LIN {X 0,Y 482.616,Z 304.958,A -85,B 0,C 180,E1 -7446.836,E2 -7446.836} C_VEL
LIN {X 0,Y 483.015,Z 308.734,A -85,B 0,C 180,E1 -7446.916,E2 -7446.916} C_VEL
LIN {X 0,Y 482.104,Z 314.511,A -85,B 0,C 180,E1 -7446.961,E2 -7446.961} C_VEL
LIN {X 0,Y 476.671,Z 329.767,A -85,B 0,C 180,E1 -7446.925,E2 -7446.925} C_VEL
LIN {X 0,Y 475.779,Z 335.739,A -85,B 0,C 180,E1 -7446.975,E2 -7446.975} C_VEL
LIN {X 0,Y 474.805,Z 416.673,A -85,B 0,C 180,E1 -7448.224,E2 -7448.224} C_VEL
LIN {X 0,Y 474.407,Z 451.66,A -85,B 0,C 180,E1 -7448.789,E2 -7448.789} C_VEL
LIN {X 0,Y 473.978,Z 467.204,A -85,B 0,C 180,E1 -7449.21,E2 -7449.21} C_VEL
LIN {X 0,Y 473.417,Z 481.814,A -85,B 0,C 180,E1 -7449.78,E2 -7449.78} C_VEL
LIN {X 0,Y 472.73,Z 495.057,A -85,B 0,C 180,E1 -7450.457,E2 -7450.457} C_VEL
LIN {X 0,Y 472.006,Z 508.633,A -85,B 0,C 180,E1 -7451.329,E2 -7451.329} C_VEL
LIN {X 0,Y 471.129,Z 521.115,A -85,B 0,C 180,E1 -7452.305,E2 -7452.305} C_VEL
LIN {X 0,Y 470.287,Z 533.744,A -85,B 0,C 180,E1 -7453.504,E2 -7453.504} C_VEL
LIN {X 0,Y 469.473,Z 545.188,A -85,B 0,C 180,E1 -7454.812,E2 -7454.812} C_VEL
LIN {X 0,Y 468.777,Z 554.815,A -85,B 0,C 180,E1 -7456.12,E2 -7456.12} C_VEL
LIN {X 0,Y 468.14,Z 563.629,A -85,B 0,C 180,E1 -7457.535,E2 -7457.535} C_VEL
LIN {X 0,Y 467.659,Z 572.092,A -85,B 0,C 180,E1 -7459.172,E2 -7459.172} C_VEL
LIN {X 0,Y 467.25,Z 579.415,A -85,B 0,C 180,E1 -7460.913,E2 -7460.913} C_VEL
LIN {X 0,Y 466.977,Z 585.225,A -85,B 0,C 180,E1 -7462.65,E2 -7462.65} C_VEL
LIN {X 0,Y 466.904,Z 588.661,A -85,B 0,C 180,E1 -7463.951,E2 -7463.951} C_VEL
LIN {X 0,Y 466.715,Z 592.15,A -85,B 0,C 180,E1 -7465.682,E2 -7465.682} C_VEL
LIN {X 0,Y 466.698,Z 594.456,A -85,B 0,C 180,E1 -7467.41,E2 -7467.41} C_VEL
LIN {X 0,Y 466.617,Z 595.638,A -85,B 0,C 180,E1 -7469.137,E2 -7469.137} C_VEL
LIN {X 0,Y 466.618,Z 595.656,A -85,B 0,C 180,E1 -7470.863,E2 -7470.863} C_VEL
LIN {X 0,Y 466.698,Z 594.543,A -85,B 0,C 180,E1 -7472.589,E2 -7472.589} C_VEL
LIN {X 0,Y 466.714,Z 592.306,A -85,B 0,C 180,E1 -7474.318,E2 -7474.318} C_VEL
LIN {X 0,Y 466.896,Z 588.882,A -85,B 0,C 180,E1 -7476.048,E2 -7476.048} C_VEL
LIN {X 0,Y 467.024,Z 584.198,A -85,B 0,C 180,E1 -7477.783,E2 -7477.783} C_VEL
LIN {X 0,Y 467.297,Z 578.125,A -85,B 0,C 180,E1 -7479.522,E2 -7479.522} C_VEL
LIN {X 0,Y 467.817,Z 570.471,A -85,B 0,C 180,E1 -7481.262,E2 -7481.262} C_VEL
LIN {X 0,Y 468.265,Z 562.094,A -85,B 0,C 180,E1 -7482.827,E2 -7482.827} C_VEL
LIN {X 0,Y 468.995,Z 552.473,A -85,B 0,C 180,E1 -7484.315,E2 -7484.315} C_VEL
LIN {X 0,Y 469.695,Z 542.383,A -85,B 0,C 180,E1 -7485.624,E2 -7485.624} C_VEL
LIN {X 0,Y 470.399,Z 532.32,A -85,B 0,C 180,E1 -7486.732,E2 -7486.732} C_VEL
LIN {X 0,Y 471.236,Z 519.597,A -85,B 0,C 180,E1 -7487.914,E2 -7487.914} C_VEL
LIN {X 0,Y 472.123,Z 506.782,A -85,B 0,C 180,E1 -7488.891,E2 -7488.891} C_VEL
LIN {X 0,Y 472.878,Z 492.726,A -85,B 0,C 180,E1 -7489.762,E2 -7489.762} C_VEL
LIN {X 0,Y 473.588,Z 477.794,A -85,B 0,C 180,E1 -7490.48,E2 -7490.48} C_VEL
LIN {X 0,Y 474.103,Z 462.506,A -85,B 0,C 180,E1 -7491.024,E2 -7491.024} C_VEL
LIN {X 0,Y 474.465,Z 448.708,A -85,B 0,C 180,E1 -7491.358,E2 -7491.358} C_VEL
LIN {X 0,Y 476.043,Z 314.849,A -85,B 0,C 180,E1 -7493.441,E2 -7493.441} C_VEL
LIN {X 0,Y 475.999,Z 305.711,A -85,B 0,C 180,E1 -7493.591,E2 -7493.591} C_VEL
LIN {X 0,Y 472.887,Z 293.254,A -85,B 0,C 180,E1 -7493.96,E2 -7493.96} C_VEL
LIN {X 0,Y 470.172,Z 286.418,A -85,B 0,C 180,E1 -7494.243,E2 -7494.243} C_VEL
LIN {X 0,Y 467.576,Z 274.869,A -85,B 0,C 180,E1 -7496.501,E2 -7496.501} C_VEL
LIN {X 0,Y 467.531,Z 274.875,A -85,B 0,C 180,E1 -7499.739,E2 -7499.739} C_VEL
LIN {X 0,Y 467.547,Z 274.874,A -85,B 0,C 180,E1 -7502.761,E2 -7502.761} C_VEL
LIN {X 0,Y 467.541,Z 274.867,A -85,B 0,C 180,E1 -7505.89,E2 -7505.89} C_VEL
LIN {X 0,Y 467.541,Z 274.873,A -85,B 0,C 180,E1 -7509.148,E2 -7509.148} C_VEL
LIN {X 0,Y 467.556,Z 274.867,A -85,B 0,C 180,E1 -7511.405,E2 -7511.405} C_VEL
LIN {X 0,Y 467.56,Z 274.87,A -85,B 0,C 180,E1 -7515.052,E2 -7515.052} C_VEL
LIN {X 0,Y 467.547,Z 274.863,A -85,B 0,C 180,E1 -7518.727,E2 -7518.727} C_VEL
LIN {X 0,Y 467.531,Z 274.868,A -85,B 0,C 180,E1 -7521.952,E2 -7521.952} C_VEL
LIN {X 0,Y 467.538,Z 274.868,A -85,B 0,C 180,E1 -7525.165,E2 -7525.165} C_VEL
LIN {X 0,Y 467.54,Z 274.871,A -85,B 0,C 180,E1 -7528.257,E2 -7528.257} C_VEL
LIN {X 0,Y 467.522,Z 274.87,A -85,B 0,C 180,E1 -7531.247,E2 -7531.247} C_VEL
LIN {X 0,Y 467.574,Z 274.868,A -85,B 0,C 180,E1 -7534.401,E2 -7534.401} C_VEL
LIN {X 0,Y 467.548,Z 274.866,A -85,B 0,C 180,E1 -7536.994,E2 -7536.994} C_VEL
LIN {X 0,Y 467.586,Z 274.862,A -85,B 0,C 180,E1 -7539.775,E2 -7539.775} C_VEL
LIN {X 0,Y 467.555,Z 274.871,A -85,B 0,C 180,E1 -7542.505,E2 -7542.505} C_VEL
LIN {X 0,Y 467.585,Z 274.858,A -85,B 0,C 180,E1 -7545.196,E2 -7545.196} C_VEL
LIN {X 0,Y 467.655,Z 274.854,A -85,B 0,C 180,E1 -7547.854,E2 -7547.854} C_VEL
LIN {X 0,Y 467.634,Z 274.851,A -85,B 0,C 180,E1 -7551.356,E2 -7551.356} C_VEL
LIN {X 0,Y 467.693,Z 274.852,A -85,B 0,C 180,E1 -7553.962,E2 -7553.962} C_VEL
LIN {X 0,Y 467.846,Z 274.828,A -85,B 0,C 180,E1 -7557.417,E2 -7557.417} C_VEL
LIN {X 0,Y 467.847,Z 274.834,A -85,B 0,C 180,E1 -7560,E2 -7560} C_VEL
LIN {X 0,Y 467.819,Z 274.835,A -85,B 0,C 180,E1 -7562.583,E2 -7562.583} C_VEL
LIN {X 0,Y 467.71,Z 274.847,A -85,B 0,C 180,E1 -7566.038,E2 -7566.038} C_VEL
LIN {X 0,Y 467.662,Z 274.853,A -85,B 0,C 180,E1 -7568.643,E2 -7568.643} C_VEL
LIN {X 0,Y 467.655,Z 274.859,A -85,B 0,C 180,E1 -7572.145,E2 -7572.145} C_VEL
LIN {X 0,Y 467.637,Z 274.855,A -85,B 0,C 180,E1 -7575.695,E2 -7575.695} C_VEL
LIN {X 0,Y 467.62,Z 274.857,A -85,B 0,C 180,E1 -7579.308,E2 -7579.308} C_VEL
LIN {X 0,Y 467.533,Z 274.873,A -85,B 0,C 180,E1 -7582.074,E2 -7582.074} C_VEL
LIN {X 0,Y 467.581,Z 274.849,A -85,B 0,C 180,E1 -7584.888,E2 -7584.888} C_VEL
LIN {X 0,Y 467.578,Z 274.865,A -85,B 0,C 180,E1 -7587.772,E2 -7587.772} C_VEL
LIN {X 0,Y 467.566,Z 274.859,A -85,B 0,C 180,E1 -7591.045,E2 -7591.045} C_VEL
LIN {X 0,Y 467.587,Z 274.864,A -85,B 0,C 180,E1 -7594.242,E2 -7594.242} C_VEL
LIN {X 0,Y 467.546,Z 274.863,A -85,B 0,C 180,E1 -7597.186,E2 -7597.186} C_VEL
LIN {X 0,Y 467.576,Z 274.864,A -85,B 0,C 180,E1 -7600.265,E2 -7600.265} C_VEL
LIN {X 0,Y 467.585,Z 274.862,A -85,B 0,C 180,E1 -7602.567,E2 -7602.567} C_VEL
LIN {X 0,Y 467.564,Z 274.866,A -85,B 0,C 180,E1 -7605.053,E2 -7605.053} C_VEL
LIN {X 0,Y 467.587,Z 274.865,A -85,B 0,C 180,E1 -7607.44,E2 -7607.44} C_VEL
LIN {X 0,Y 467.581,Z 274.864,A -85,B 0,C 180,E1 -7610.855,E2 -7610.855} C_VEL
LIN {X 0,Y 467.561,Z 274.868,A -85,B 0,C 180,E1 -7614.261,E2 -7614.261} C_VEL
LIN {X 0,Y 467.581,Z 274.868,A -85,B 0,C 180,E1 -7617.321,E2 -7617.321} C_VEL
LIN {X 0,Y 467.582,Z 274.98,A -85,B 0,C 180,E1 -7619.153,E2 -7619.153} C_VEL
LIN {X 0,Y 471.016,Z 288.782,A -85,B 0,C 180,E1 -7621.48,E2 -7621.48} C_VEL
LIN {X 0,Y 472.395,Z 295.297,A -85,B 0,C 180,E1 -7622.536,E2 -7622.536} C_VEL
LIN {X 0,Y 471.328,Z 315.414,A -85,B 0,C 180,E1 -7625.446,E2 -7625.446} C_VEL
LIN {X 0,Y 471.122,Z 318.255,A -85,B 0,C 180,E1 -7625.853,E2 -7625.853} C_VEL
LIN {X 0,Y 475.844,Z 343.181,A -85,B 0,C 180,E1 -7626.514,E2 -7626.514} C_VEL
LIN {X 0,Y 474.196,Z 484.206,A -85,B 0,C 180,E1 -7628.709,E2 -7628.709} C_VEL
LIN {X 0,Y 473.7,Z 499.79,A -85,B 0,C 180,E1 -7629.113,E2 -7629.113} C_VEL
LIN {X 0,Y 473.008,Z 515.238,A -85,B 0,C 180,E1 -7629.698,E2 -7629.698} C_VEL
LIN {X 0,Y 472.193,Z 529.814,A -85,B 0,C 180,E1 -7630.435,E2 -7630.435} C_VEL
LIN {X 0,Y 471.378,Z 543.34,A -85,B 0,C 180,E1 -7631.304,E2 -7631.304} C_VEL
LIN {X 0,Y 470.541,Z 555.818,A -85,B 0,C 180,E1 -7632.283,E2 -7632.283} C_VEL
LIN {X 0,Y 469.628,Z 568.514,A -85,B 0,C 180,E1 -7633.481,E2 -7633.481} C_VEL
LIN {X 0,Y 468.867,Z 580.057,A -85,B 0,C 180,E1 -7634.793,E2 -7634.793} C_VEL
LIN {X 0,Y 468.278,Z 589.779,A -85,B 0,C 180,E1 -7636.106,E2 -7636.106} C_VEL
LIN {X 0,Y 467.631,Z 599.448,A -85,B 0,C 180,E1 -7637.655,E2 -7637.655} C_VEL
LIN {X 0,Y 467.34,Z 607.294,A -85,B 0,C 180,E1 -7639.166,E2 -7639.166} C_VEL
LIN {X 0,Y 466.956,Z 614.727,A -85,B 0,C 180,E1 -7640.908,E2 -7640.908} C_VEL
LIN {X 0,Y 466.811,Z 620.631,A -85,B 0,C 180,E1 -7642.648,E2 -7642.648} C_VEL
LIN {X 0,Y 466.705,Z 624.139,A -85,B 0,C 180,E1 -7643.95,E2 -7643.95} C_VEL
LIN {X 0,Y 466.616,Z 627.685,A -85,B 0,C 180,E1 -7645.681,E2 -7645.681} C_VEL
LIN {X 0,Y 466.656,Z 630.021,A -85,B 0,C 180,E1 -7647.411,E2 -7647.411} C_VEL
LIN {X 0,Y 466.617,Z 631.194,A -85,B 0,C 180,E1 -7649.137,E2 -7649.137} C_VEL
LIN {X 0,Y 466.617,Z 631.193,A -85,B 0,C 180,E1 -7650.863,E2 -7650.863} C_VEL
LIN {X 0,Y 466.656,Z 630.016,A -85,B 0,C 180,E1 -7652.59,E2 -7652.59} C_VEL
LIN {X 0,Y 466.616,Z 627.679,A -85,B 0,C 180,E1 -7654.319,E2 -7654.319} C_VEL
LIN {X 0,Y 466.696,Z 624.137,A -85,B 0,C 180,E1 -7656.051,E2 -7656.051} C_VEL
LIN {X 0,Y 466.827,Z 619.299,A -85,B 0,C 180,E1 -7657.788,E2 -7657.788} C_VEL
LIN {X 0,Y 467.001,Z 613.033,A -85,B 0,C 180,E1 -7659.529,E2 -7659.529} C_VEL
LIN {X 0,Y 467.41,Z 605.171,A -85,B 0,C 180,E1 -7661.273,E2 -7661.273} C_VEL
LIN {X 0,Y 467.842,Z 596.762,A -85,B 0,C 180,E1 -7662.81,E2 -7662.81} C_VEL
LIN {X 0,Y 468.466,Z 586.744,A -85,B 0,C 180,E1 -7664.332,E2 -7664.332} C_VEL
LIN {X 0,Y 469.144,Z 576.454,A -85,B 0,C 180,E1 -7665.644,E2 -7665.644} C_VEL
LIN {X 0,Y 470.042,Z 564.048,A -85,B 0,C 180,E1 -7666.968,E2 -7666.968} C_VEL
LIN {X 0,Y 470.895,Z 550.568,A -85,B 0,C 180,E1 -7668.153,E2 -7668.153} C_VEL
LIN {X 0,Y 471.779,Z 536.906,A -85,B 0,C 180,E1 -7669.132,E2 -7669.132} C_VEL
LIN {X 0,Y 472.584,Z 522.762,A -85,B 0,C 180,E1 -7669.945,E2 -7669.945} C_VEL
LIN {X 0,Y 473.305,Z 507.927,A -85,B 0,C 180,E1 -7670.605,E2 -7670.605} C_VEL
LIN {X 0,Y 473.946,Z 492.295,A -85,B 0,C 180,E1 -7671.104,E2 -7671.104} C_VEL
LIN {X 0,Y 474.32,Z 476.367,A -85,B 0,C 180,E1 -7671.428,E2 -7671.428} C_VEL
LIN {X 0,Y 475.826,Z 343.138,A -85,B 0,C 180,E1 -7673.485,E2 -7673.485} C_VEL
LIN {X 0,Y 471.104,Z 318.257,A -85,B 0,C 180,E1 -7674.145,E2 -7674.145} C_VEL
LIN {X 0,Y 472.319,Z 298.282,A -85,B 0,C 180,E1 -7677.022,E2 -7677.022} C_VEL
LIN {X 0,Y 472.405,Z 295.266,A -85,B 0,C 180,E1 -7677.464,E2 -7677.464} C_VEL
LIN {X 0,Y 469.063,Z 280.585,A -85,B 0,C 180,E1 -7679.88,E2 -7679.88} C_VEL
LIN {X 0,Y 467.56,Z 274.867,A -85,B 0,C 180,E1 -7680.878,E2 -7680.878} C_VEL
LIN {X 0,Y 467.588,Z 274.866,A -85,B 0,C 180,E1 -7683.789,E2 -7683.789} C_VEL
LIN {X 0,Y 467.55,Z 274.867,A -85,B 0,C 180,E1 -7687.187,E2 -7687.187} C_VEL
LIN {X 0,Y 467.574,Z 274.863,A -85,B 0,C 180,E1 -7690.266,E2 -7690.266} C_VEL
LIN {X 0,Y 467.551,Z 274.867,A -85,B 0,C 180,E1 -7693.746,E2 -7693.746} C_VEL
LIN {X 0,Y 467.554,Z 274.865,A -85,B 0,C 180,E1 -7696.255,E2 -7696.255} C_VEL
LIN {X 0,Y 467.581,Z 274.865,A -85,B 0,C 180,E1 -7698.724,E2 -7698.724} C_VEL
LIN {X 0,Y 467.565,Z 274.868,A -85,B 0,C 180,E1 -7701.956,E2 -7701.956} C_VEL
LIN {X 0,Y 467.566,Z 274.862,A -85,B 0,C 180,E1 -7705.168,E2 -7705.168} C_VEL
LIN {X 0,Y 467.587,Z 274.865,A -85,B 0,C 180,E1 -7708.26,E2 -7708.26} C_VEL
LIN {X 0,Y 467.559,Z 274.862,A -85,B 0,C 180,E1 -7711.249,E2 -7711.249} C_VEL
LIN {X 0,Y 467.584,Z 274.864,A -85,B 0,C 180,E1 -7714.159,E2 -7714.159} C_VEL
LIN {X 0,Y 467.58,Z 274.858,A -85,B 0,C 180,E1 -7716.996,E2 -7716.996} C_VEL
LIN {X 0,Y 467.626,Z 274.86,A -85,B 0,C 180,E1 -7719.777,E2 -7719.777} C_VEL
LIN {X 0,Y 467.6,Z 274.863,A -85,B 0,C 180,E1 -7722.507,E2 -7722.507} C_VEL
LIN {X 0,Y 467.609,Z 274.856,A -85,B 0,C 180,E1 -7725.197,E2 -7725.197} C_VEL
LIN {X 0,Y 467.662,Z 274.858,A -85,B 0,C 180,E1 -7727.855,E2 -7727.855} C_VEL
LIN {X 0,Y 467.662,Z 274.854,A -85,B 0,C 180,E1 -7731.357,E2 -7731.357} C_VEL
LIN {X 0,Y 467.708,Z 274.851,A -85,B 0,C 180,E1 -7733.962,E2 -7733.962} C_VEL
LIN {X 0,Y 467.818,Z 274.832,A -85,B 0,C 180,E1 -7737.417,E2 -7737.417} C_VEL
LIN {X 0,Y 467.854,Z 274.833,A -85,B 0,C 180,E1 -7740,E2 -7740} C_VEL
LIN {X 0,Y 467.827,Z 274.831,A -85,B 0,C 180,E1 -7742.583,E2 -7742.583} C_VEL
LIN {X 0,Y 467.699,Z 274.849,A -85,B 0,C 180,E1 -7746.038,E2 -7746.038} C_VEL
LIN {X 0,Y 467.64,Z 274.855,A -85,B 0,C 180,E1 -7748.644,E2 -7748.644} C_VEL
LIN {X 0,Y 467.661,Z 274.855,A -85,B 0,C 180,E1 -7752.145,E2 -7752.145} C_VEL
LIN {X 0,Y 467.617,Z 274.862,A -85,B 0,C 180,E1 -7755.696,E2 -7755.696} C_VEL
LIN {X 0,Y 467.577,Z 274.86,A -85,B 0,C 180,E1 -7758.748,E2 -7758.748} C_VEL
LIN {X 0,Y 467.563,Z 274.869,A -85,B 0,C 180,E1 -7761.261,E2 -7761.261} C_VEL
LIN {X 0,Y 467.552,Z 274.869,A -85,B 0,C 180,E1 -7763.945,E2 -7763.945} C_VEL
LIN {X 0,Y 467.529,Z 274.865,A -85,B 0,C 180,E1 -7766.806,E2 -7766.806} C_VEL
LIN {X 0,Y 467.513,Z 274.873,A -85,B 0,C 180,E1 -7769.741,E2 -7769.741} C_VEL
LIN {X 0,Y 467.551,Z 274.866,A -85,B 0,C 180,E1 -7772.761,E2 -7772.761} C_VEL
LIN {X 0,Y 467.541,Z 274.868,A -85,B 0,C 180,E1 -7775.891,E2 -7775.891} C_VEL
LIN {X 0,Y 467.529,Z 274.871,A -85,B 0,C 180,E1 -7779.15,E2 -7779.15} C_VEL
LIN {X 0,Y 467.552,Z 274.87,A -85,B 0,C 180,E1 -7781.406,E2 -7781.406} C_VEL
LIN {X 0,Y 467.532,Z 274.871,A -85,B 0,C 180,E1 -7784.952,E2 -7784.952} C_VEL
LIN {X 0,Y 467.55,Z 274.866,A -85,B 0,C 180,E1 -7788.594,E2 -7788.594} C_VEL
LIN {X 0,Y 467.535,Z 274.868,A -85,B 0,C 180,E1 -7791.952,E2 -7791.952} C_VEL
LIN {X 0,Y 467.543,Z 274.87,A -85,B 0,C 180,E1 -7795.165,E2 -7795.165} C_VEL
LIN {X 0,Y 467.544,Z 274.867,A -85,B 0,C 180,E1 -7798.256,E2 -7798.256} C_VEL
LIN {X 0,Y 467.527,Z 274.876,A -85,B 0,C 180,E1 -7801.247,E2 -7801.247} C_VEL
LIN {X 0,Y 467.57,Z 274.908,A -85,B 0,C 180,E1 -7803.618,E2 -7803.618} C_VEL
LIN {X 0,Y 470.221,Z 286.501,A -85,B 0,C 180,E1 -7805.868,E2 -7805.868} C_VEL
LIN {X 0,Y 473.542,Z 295.441,A -85,B 0,C 180,E1 -7806.204,E2 -7806.204} C_VEL
LIN {X 0,Y 476.129,Z 307.183,A -85,B 0,C 180,E1 -7806.532,E2 -7806.532} C_VEL
LIN {X 0,Y 475.779,Z 335.739,A -85,B 0,C 180,E1 -7806.975,E2 -7806.975} C_VEL
LIN {X 0,Y 475.114,Z 341.592,A -85,B 0,C 180,E1 -7807.034,E2 -7807.034} C_VEL
LIN {X 0,Y 469.576,Z 360.655,A -85,B 0,C 180,E1 -7807.055,E2 -7807.055} C_VEL
LIN {X 0,Y 468.938,Z 366.506,A -85,B 0,C 180,E1 -7807.117,E2 -7807.117} C_VEL
LIN {X 0,Y 467.811,Z 451.948,A -85,B 0,C 180,E1 -7808.475,E2 -7808.475} C_VEL
LIN {X 0,Y 467.371,Z 467.458,A -85,B 0,C 180,E1 -7808.902,E2 -7808.902} C_VEL
LIN {X 0,Y 466.758,Z 482.247,A -85,B 0,C 180,E1 -7809.486,E2 -7809.486} C_VEL
LIN {X 0,Y 465.949,Z 497.227,A -85,B 0,C 180,E1 -7810.276,E2 -7810.276} C_VEL
LIN {X 0,Y 465.169,Z 510.471,A -85,B 0,C 180,E1 -7811.158,E2 -7811.158} C_VEL
LIN {X 0,Y 464.218,Z 523.927,A -85,B 0,C 180,E1 -7812.261,E2 -7812.261} C_VEL
LIN {X 0,Y 463.314,Z 536.125,A -85,B 0,C 180,E1 -7813.475,E2 -7813.475} C_VEL
LIN {X 0,Y 462.476,Z 547.228,A -85,B 0,C 180,E1 -7814.802,E2 -7814.802} C_VEL
LIN {X 0,Y 461.647,Z 558.012,A -85,B 0,C 180,E1 -7816.351,E2 -7816.351} C_VEL
LIN {X 0,Y 461.053,Z 566.951,A -85,B 0,C 180,E1 -7817.901,E2 -7817.901} C_VEL
LIN {X 0,Y 460.499,Z 574.361,A -85,B 0,C 180,E1 -7819.447,E2 -7819.447} C_VEL
LIN {X 0,Y 460.137,Z 581.283,A -85,B 0,C 180,E1 -7821.214,E2 -7821.214} C_VEL
LIN {X 0,Y 459.849,Z 586.724,A -85,B 0,C 180,E1 -7822.977,E2 -7822.977} C_VEL
LIN {X 0,Y 459.701,Z 590.83,A -85,B 0,C 180,E1 -7824.736,E2 -7824.736} C_VEL
LIN {X 0,Y 459.683,Z 593.715,A -85,B 0,C 180,E1 -7826.493,E2 -7826.493} C_VEL
LIN {X 0,Y 459.571,Z 595.456,A -85,B 0,C 180,E1 -7828.247,E2 -7828.247} C_VEL
LIN {X 0,Y 459.528,Z 596.066,A -85,B 0,C 180,E1 -7830,E2 -7830} C_VEL
LIN {X 0,Y 459.572,Z 595.508,A -85,B 0,C 180,E1 -7831.752,E2 -7831.752} C_VEL
LIN {X 0,Y 459.683,Z 593.836,A -85,B 0,C 180,E1 -7833.506,E2 -7833.506} C_VEL
LIN {X 0,Y 459.697,Z 591.017,A -85,B 0,C 180,E1 -7835.263,E2 -7835.263} C_VEL
LIN {X 0,Y 459.844,Z 586.976,A -85,B 0,C 180,E1 -7837.023,E2 -7837.023} C_VEL
LIN {X 0,Y 460.125,Z 581.614,A -85,B 0,C 180,E1 -7838.785,E2 -7838.785} C_VEL
LIN {X 0,Y 460.474,Z 574.782,A -85,B 0,C 180,E1 -7840.553,E2 -7840.553} C_VEL
LIN {X 0,Y 461.015,Z 567.425,A -85,B 0,C 180,E1 -7842.099,E2 -7842.099} C_VEL
LIN {X 0,Y 461.626,Z 558.564,A -85,B 0,C 180,E1 -7843.649,E2 -7843.649} C_VEL
LIN {X 0,Y 462.294,Z 549.524,A -85,B 0,C 180,E1 -7844.977,E2 -7844.977} C_VEL
LIN {X 0,Y 463.106,Z 538.855,A -85,B 0,C 180,E1 -7846.305,E2 -7846.305} C_VEL
LIN {X 0,Y 463.984,Z 527.536,A -85,B 0,C 180,E1 -7847.488,E2 -7847.488} C_VEL
LIN {X 0,Y 464.895,Z 514.473,A -85,B 0,C 180,E1 -7848.624,E2 -7848.624} C_VEL
LIN {X 0,Y 465.793,Z 500.42,A -85,B 0,C 180,E1 -7849.616,E2 -7849.616} C_VEL
LIN {X 0,Y 466.545,Z 487.148,A -85,B 0,C 180,E1 -7850.365,E2 -7850.365} C_VEL
LIN {X 0,Y 467.176,Z 472.197,A -85,B 0,C 180,E1 -7851.02,E2 -7851.02} C_VEL
LIN {X 0,Y 467.672,Z 457.345,A -85,B 0,C 180,E1 -7851.487,E2 -7851.487} C_VEL
LIN {X 0,Y 468.002,Z 442.394,A -85,B 0,C 180,E1 -7851.789,E2 -7851.789} C_VEL
LIN {X 0,Y 469.559,Z 315.136,A -85,B 0,C 180,E1 -7853.783,E2 -7853.783} C_VEL
LIN {X 0,Y 469.469,Z 306.681,A -85,B 0,C 180,E1 -7853.927,E2 -7853.927} C_VEL
LIN {X 0,Y 466.833,Z 296.114,A -85,B 0,C 180,E1 -7854.247,E2 -7854.247} C_VEL
LIN {X 0,Y 463.026,Z 286.71,A -85,B 0,C 180,E1 -7854.64,E2 -7854.64} C_VEL
LIN {X 0,Y 460.504,Z 275.751,A -85,B 0,C 180,E1 -7856.818,E2 -7856.818} C_VEL
LIN {X 0,Y 460.509,Z 275.751,A -85,B 0,C 180,E1 -7859.553,E2 -7859.553} C_VEL
LIN {X 0,Y 460.5,Z 275.75,A -85,B 0,C 180,E1 -7862.924,E2 -7862.924} C_VEL
LIN {X 0,Y 460.484,Z 275.746,A -85,B 0,C 180,E1 -7866.012,E2 -7866.012} C_VEL
LIN {X 0,Y 460.49,Z 275.753,A -85,B 0,C 180,E1 -7868.889,E2 -7868.889} C_VEL
LIN {X 0,Y 460.5,Z 275.745,A -85,B 0,C 180,E1 -7871.598,E2 -7871.598} C_VEL
LIN {X 0,Y 460.508,Z 275.745,A -85,B 0,C 180,E1 -7874.589,E2 -7874.589} C_VEL
LIN {X 0,Y 460.468,Z 275.738,A -85,B 0,C 180,E1 -7877.812,E2 -7877.812} C_VEL
LIN {X 0,Y 460.472,Z 275.749,A -85,B 0,C 180,E1 -7880.131,E2 -7880.131} C_VEL
LIN {X 0,Y 460.452,Z 275.736,A -85,B 0,C 180,E1 -7883.468,E2 -7883.468} C_VEL
LIN {X 0,Y 460.498,Z 275.752,A -85,B 0,C 180,E1 -7886.672,E2 -7886.672} C_VEL
LIN {X 0,Y 460.476,Z 275.746,A -85,B 0,C 180,E1 -7889.757,E2 -7889.757} C_VEL
LIN {X 0,Y 460.485,Z 275.749,A -85,B 0,C 180,E1 -7892.75,E2 -7892.75} C_VEL
LIN {X 0,Y 460.509,Z 275.743,A -85,B 0,C 180,E1 -7895.666,E2 -7895.666} C_VEL
LIN {X 0,Y 460.512,Z 275.75,A -85,B 0,C 180,E1 -7898.581,E2 -7898.581} C_VEL
LIN {X 0,Y 460.533,Z 275.735,A -85,B 0,C 180,E1 -7901.308,E2 -7901.308} C_VEL
LIN {X 0,Y 460.544,Z 275.737,A -85,B 0,C 180,E1 -7904.964,E2 -7904.964} C_VEL
LIN {X 0,Y 460.606,Z 275.736,A -85,B 0,C 180,E1 -7908.559,E2 -7908.559} C_VEL
LIN {X 0,Y 460.621,Z 275.73,A -85,B 0,C 180,E1 -7912.107,E2 -7912.107} C_VEL
LIN {X 0,Y 460.669,Z 275.722,A -85,B 0,C 180,E1 -7914.748,E2 -7914.748} C_VEL
LIN {X 0,Y 460.786,Z 275.707,A -85,B 0,C 180,E1 -7917.377,E2 -7917.377} C_VEL
LIN {X 0,Y 460.817,Z 275.709,A -85,B 0,C 180,E1 -7920,E2 -7920} C_VEL
LIN {X 0,Y 460.763,Z 275.714,A -85,B 0,C 180,E1 -7922.623,E2 -7922.623} C_VEL
LIN {X 0,Y 460.675,Z 275.723,A -85,B 0,C 180,E1 -7926.13,E2 -7926.13} C_VEL
LIN {X 0,Y 460.613,Z 275.731,A -85,B 0,C 180,E1 -7928.776,E2 -7928.776} C_VEL
LIN {X 0,Y 460.612,Z 275.734,A -85,B 0,C 180,E1 -7932.445,E2 -7932.445} C_VEL
LIN {X 0,Y 460.599,Z 275.735,A -85,B 0,C 180,E1 -7935.997,E2 -7935.997} C_VEL
LIN {X 0,Y 460.566,Z 275.737,A -85,B 0,C 180,E1 -7939.616,E2 -7939.616} C_VEL
LIN {X 0,Y 460.509,Z 275.744,A -85,B 0,C 180,E1 -7942.429,E2 -7942.429} C_VEL
LIN {X 0,Y 460.547,Z 275.728,A -85,B 0,C 180,E1 -7945.797,E2 -7945.797} C_VEL
LIN {X 0,Y 460.525,Z 275.745,A -85,B 0,C 180,E1 -7948.235,E2 -7948.235} C_VEL
LIN {X 0,Y 460.519,Z 275.738,A -85,B 0,C 180,E1 -7951.283,E2 -7951.283} C_VEL
LIN {X 0,Y 460.531,Z 275.741,A -85,B 0,C 180,E1 -7954.506,E2 -7954.506} C_VEL
LIN {X 0,Y 460.499,Z 275.74,A -85,B 0,C 180,E1 -7957.623,E2 -7957.623} C_VEL
LIN {X 0,Y 460.54,Z 275.741,A -85,B 0,C 180,E1 -7960.27,E2 -7960.27} C_VEL
LIN {X 0,Y 460.497,Z 275.749,A -85,B 0,C 180,E1 -7963.376,E2 -7963.376} C_VEL
LIN {X 0,Y 460.497,Z 275.744,A -85,B 0,C 180,E1 -7966.625,E2 -7966.625} C_VEL
LIN {X 0,Y 460.54,Z 275.74,A -85,B 0,C 180,E1 -7969.731,E2 -7969.731} C_VEL
LIN {X 0,Y 460.499,Z 275.745,A -85,B 0,C 180,E1 -7972.524,E2 -7972.524} C_VEL
LIN {X 0,Y 460.547,Z 275.743,A -85,B 0,C 180,E1 -7975.624,E2 -7975.624} C_VEL
LIN {X 0,Y 460.55,Z 275.859,A -85,B 0,C 180,E1 -7978.81,E2 -7978.81} C_VEL
LIN {X 0,Y 464.005,Z 289.714,A -85,B 0,C 180,E1 -7981.194,E2 -7981.194} C_VEL
LIN {X 0,Y 465.531,Z 296.646,A -85,B 0,C 180,E1 -7982.341,E2 -7982.341} C_VEL
LIN {X 0,Y 464.653,Z 314.306,A -85,B 0,C 180,E1 -7984.944,E2 -7984.944} C_VEL
LIN {X 0,Y 464.355,Z 317.975,A -85,B 0,C 180,E1 -7985.477,E2 -7985.477} C_VEL
LIN {X 0,Y 469.371,Z 345.068,A -85,B 0,C 180,E1 -7986.206,E2 -7986.206} C_VEL
LIN {X 0,Y 467.544,Z 485.275,A -85,B 0,C 180,E1 -7988.42,E2 -7988.42} C_VEL
LIN {X 0,Y 466.978,Z 501.269,A -85,B 0,C 180,E1 -7988.859,E2 -7988.859} C_VEL
LIN {X 0,Y 466.301,Z 515.516,A -85,B 0,C 180,E1 -7989.418,E2 -7989.418} C_VEL
LIN {X 0,Y 465.468,Z 529.546,A -85,B 0,C 180,E1 -7990.14,E2 -7990.14} C_VEL
LIN {X 0,Y 464.615,Z 543.071,A -85,B 0,C 180,E1 -7991.021,E2 -7991.021} C_VEL
LIN {X 0,Y 463.681,Z 555.546,A -85,B 0,C 180,E1 -7992.012,E2 -7992.012} C_VEL
LIN {X 0,Y 462.854,Z 566.577,A -85,B 0,C 180,E1 -7993.057,E2 -7993.057} C_VEL
LIN {X 0,Y 462.08,Z 577.99,A -85,B 0,C 180,E1 -7994.338,E2 -7994.338} C_VEL
LIN {X 0,Y 461.4,Z 588.008,A -85,B 0,C 180,E1 -7995.67,E2 -7995.67} C_VEL
LIN {X 0,Y 460.795,Z 596.68,A -85,B 0,C 180,E1 -7997.022,E2 -7997.022} C_VEL
LIN {X 0,Y 460.354,Z 604.91,A -85,B 0,C 180,E1 -7998.553,E2 -7998.553} C_VEL
LIN {X 0,Y 460.057,Z 610.943,A -85,B 0,C 180,E1 -7999.882,E2 -7999.882} C_VEL
LIN {X 0,Y 459.783,Z 617.587,A -85,B 0,C 180,E1 -8001.651,E2 -8001.651} C_VEL
LIN {X 0,Y 459.664,Z 621.615,A -85,B 0,C 180,E1 -8002.975,E2 -8002.975} C_VEL
LIN {X 0,Y 459.594,Z 625.798,A -85,B 0,C 180,E1 -8004.736,E2 -8004.736} C_VEL
LIN {X 0,Y 459.568,Z 628.731,A -85,B 0,C 180,E1 -8006.493,E2 -8006.493} C_VEL
LIN {X 0,Y 459.539,Z 630.48,A -85,B 0,C 180,E1 -8008.248,E2 -8008.248} C_VEL
LIN {X 0,Y 459.527,Z 631.079,A -85,B 0,C 180,E1 -8010,E2 -8010} C_VEL
LIN {X 0,Y 459.539,Z 630.477,A -85,B 0,C 180,E1 -8011.753,E2 -8011.753} C_VEL
LIN {X 0,Y 459.568,Z 628.725,A -85,B 0,C 180,E1 -8013.507,E2 -8013.507} C_VEL
LIN {X 0,Y 459.592,Z 625.793,A -85,B 0,C 180,E1 -8015.265,E2 -8015.265} C_VEL
LIN {X 0,Y 459.652,Z 621.615,A -85,B 0,C 180,E1 -8017.026,E2 -8017.026} C_VEL
LIN {X 0,Y 459.836,Z 616.081,A -85,B 0,C 180,E1 -8018.792,E2 -8018.792} C_VEL
LIN {X 0,Y 460.198,Z 609.044,A -85,B 0,C 180,E1 -8020.56,E2 -8020.56} C_VEL
LIN {X 0,Y 460.582,Z 600.285,A -85,B 0,C 180,E1 -8022.335,E2 -8022.335} C_VEL
LIN {X 0,Y 461.191,Z 590.991,A -85,B 0,C 180,E1 -8023.888,E2 -8023.888} C_VEL
LIN {X 0,Y 461.83,Z 581.544,A -85,B 0,C 180,E1 -8025.219,E2 -8025.219} C_VEL
LIN {X 0,Y 462.735,Z 569.304,A -85,B 0,C 180,E1 -8026.659,E2 -8026.659} C_VEL
LIN {X 0,Y 463.629,Z 556.827,A -85,B 0,C 180,E1 -8027.877,E2 -8027.877} C_VEL
LIN {X 0,Y 464.521,Z 544.557,A -85,B 0,C 180,E1 -8028.869,E2 -8028.869} C_VEL
LIN {X 0,Y 465.388,Z 531.312,A -85,B 0,C 180,E1 -8029.749,E2 -8029.749} C_VEL
LIN {X 0,Y 466.212,Z 517.055,A -85,B 0,C 180,E1 -8030.506,E2 -8030.506} C_VEL
LIN {X 0,Y 466.89,Z 502.902,A -85,B 0,C 180,E1 -8031.081,E2 -8031.081} C_VEL
LIN {X 0,Y 467.471,Z 487.442,A -85,B 0,C 180,E1 -8031.527,E2 -8031.527} C_VEL
LIN {X 0,Y 467.826,Z 465.331,A -85,B 0,C 180,E1 -8031.915,E2 -8031.915} C_VEL
LIN {X 0,Y 469.256,Z 343.824,A -85,B 0,C 180,E1 -8033.818,E2 -8033.818} C_VEL
LIN {X 0,Y 464.329,Z 317.858,A -85,B 0,C 180,E1 -8034.539,E2 -8034.539} C_VEL
LIN {X 0,Y 465.558,Z 298.23,A -85,B 0,C 180,E1 -8037.415,E2 -8037.415} C_VEL
LIN {X 0,Y 465.223,Z 294.982,A -85,B 0,C 180,E1 -8037.925,E2 -8037.925} C_VEL
LIN {X 0,Y 461.678,Z 280.296,A -85,B 0,C 180,E1 -8040.409,E2 -8040.409} C_VEL
LIN {X 0,Y 460.527,Z 275.742,A -85,B 0,C 180,E1 -8041.225,E2 -8041.225} C_VEL
LIN {X 0,Y 460.534,Z 275.747,A -85,B 0,C 180,E1 -8044.506,E2 -8044.506} C_VEL
LIN {X 0,Y 460.503,Z 275.745,A -85,B 0,C 180,E1 -8047.624,E2 -8047.624} C_VEL
LIN {X 0,Y 460.539,Z 275.739,A -85,B 0,C 180,E1 -8050.269,E2 -8050.269} C_VEL
LIN {X 0,Y 460.511,Z 275.743,A -85,B 0,C 180,E1 -8053.375,E2 -8053.375} C_VEL
LIN {X 0,Y 460.499,Z 275.743,A -85,B 0,C 180,E1 -8056.625,E2 -8056.625} C_VEL
LIN {X 0,Y 460.542,Z 275.74,A -85,B 0,C 180,E1 -8059.732,E2 -8059.732} C_VEL
LIN {X 0,Y 460.5,Z 275.749,A -85,B 0,C 180,E1 -8062.525,E2 -8062.525} C_VEL
LIN {X 0,Y 460.549,Z 275.737,A -85,B 0,C 180,E1 -8065.624,E2 -8065.624} C_VEL
LIN {X 0,Y 460.541,Z 275.74,A -85,B 0,C 180,E1 -8068.745,E2 -8068.745} C_VEL
LIN {X 0,Y 460.555,Z 275.742,A -85,B 0,C 180,E1 -8072.262,E2 -8072.262} C_VEL
LIN {X 0,Y 460.538,Z 275.74,A -85,B 0,C 180,E1 -8074.704,E2 -8074.704} C_VEL
LIN {X 0,Y 460.515,Z 275.74,A -85,B 0,C 180,E1 -8077.572,E2 -8077.572} C_VEL
LIN {X 0,Y 460.572,Z 275.735,A -85,B 0,C 180,E1 -8080.385,E2 -8080.385} C_VEL
LIN {X 0,Y 460.609,Z 275.734,A -85,B 0,C 180,E1 -8084.059,E2 -8084.059} C_VEL
LIN {X 0,Y 460.615,Z 275.734,A -85,B 0,C 180,E1 -8087.666,E2 -8087.666} C_VEL
LIN {X 0,Y 460.614,Z 275.731,A -85,B 0,C 180,E1 -8091.224,E2 -8091.224} C_VEL
LIN {X 0,Y 460.674,Z 275.725,A -85,B 0,C 180,E1 -8093.87,E2 -8093.87} C_VEL
LIN {X 0,Y 460.762,Z 275.711,A -85,B 0,C 180,E1 -8097.377,E2 -8097.377} C_VEL
LIN {X 0,Y 460.823,Z 275.708,A -85,B 0,C 180,E1 -8100,E2 -8100} C_VEL
LIN {X 0,Y 460.772,Z 275.71,A -85,B 0,C 180,E1 -8102.623,E2 -8102.623} C_VEL
LIN {X 0,Y 460.665,Z 275.724,A -85,B 0,C 180,E1 -8106.131,E2 -8106.131} C_VEL
LIN {X 0,Y 460.595,Z 275.733,A -85,B 0,C 180,E1 -8108.777,E2 -8108.777} C_VEL
LIN {X 0,Y 460.614,Z 275.731,A -85,B 0,C 180,E1 -8112.334,E2 -8112.334} C_VEL
LIN {X 0,Y 460.562,Z 275.741,A -85,B 0,C 180,E1 -8115.978,E2 -8115.978} C_VEL
LIN {X 0,Y 460.535,Z 275.737,A -85,B 0,C 180,E1 -8118.886,E2 -8118.886} C_VEL
LIN {X 0,Y 460.513,Z 275.749,A -85,B 0,C 180,E1 -8121.486,E2 -8121.486} C_VEL
LIN {X 0,Y 460.514,Z 275.743,A -85,B 0,C 180,E1 -8124.334,E2 -8124.334} C_VEL
LIN {X 0,Y 460.488,Z 275.741,A -85,B 0,C 180,E1 -8127.249,E2 -8127.249} C_VEL
LIN {X 0,Y 460.482,Z 275.746,A -85,B 0,C 180,E1 -8130.242,E2 -8130.242} C_VEL
LIN {X 0,Y 460.503,Z 275.747,A -85,B 0,C 180,E1 -8133.327,E2 -8133.327} C_VEL
LIN {X 0,Y 460.458,Z 275.748,A -85,B 0,C 180,E1 -8136.531,E2 -8136.531} C_VEL
LIN {X 0,Y 460.477,Z 275.749,A -85,B 0,C 180,E1 -8139.868,E2 -8139.868} C_VEL
LIN {X 0,Y 460.458,Z 275.752,A -85,B 0,C 180,E1 -8142.892,E2 -8142.892} C_VEL
LIN {X 0,Y 460.481,Z 275.747,A -85,B 0,C 180,E1 -8145.834,E2 -8145.834} C_VEL
LIN {X 0,Y 460.501,Z 275.748,A -85,B 0,C 180,E1 -8148.985,E2 -8148.985} C_VEL
LIN {X 0,Y 460.48,Z 275.746,A -85,B 0,C 180,E1 -8152.374,E2 -8152.374} C_VEL
LIN {X 0,Y 460.524,Z 275.74,A -85,B 0,C 180,E1 -8155.621,E2 -8155.621} C_VEL
LIN {X 0,Y 460.506,Z 275.745,A -85,B 0,C 180,E1 -8158.742,E2 -8158.742} C_VEL
LIN {X 0,Y 460.497,Z 275.749,A -85,B 0,C 180,E1 -8161.763,E2 -8161.763} C_VEL
LIN {X 0,Y 460.509,Z 275.832,A -85,B 0,C 180,E1 -8163.303,E2 -8163.303} C_VEL
LIN {X 0,Y 463.1,Z 286.999,A -85,B 0,C 180,E1 -8165.483,E2 -8165.483} C_VEL
LIN {X 0,Y 467.347,Z 297.823,A -85,B 0,C 180,E1 -8165.903,E2 -8165.903} C_VEL
LIN {X 0,Y 469.638,Z 307.787,A -85,B 0,C 180,E1 -8166.193,E2 -8166.193} C_VEL
LIN {X 0,Y 468.938,Z 366.506,A -85,B 0,C 180,E1 -8167.117,E2 -8167.117} C_VEL
LIN {X 0,Y 468.312,Z 372.352,A -85,B 0,C 180,E1 -8167.179,E2 -8167.179} C_VEL
LIN {X 0,Y 462.791,Z 391.409,A -85,B 0,C 180,E1 -8167.203,E2 -8167.203} C_VEL
LIN {X 0,Y 462.062,Z 397.262,A -85,B 0,C 180,E1 -8167.261,E2 -8167.261} C_VEL
LIN {X 0,Y 461.213,Z 452.539,A -85,B 0,C 180,E1 -8168.159,E2 -8168.159} C_VEL
LIN {X 0,Y 460.77,Z 467.466,A -85,B 0,C 180,E1 -8168.574,E2 -8168.574} C_VEL
LIN {X 0,Y 460.154,Z 481.74,A -85,B 0,C 180,E1 -8169.141,E2 -8169.141} C_VEL
LIN {X 0,Y 459.384,Z 495.613,A -85,B 0,C 180,E1 -8169.865,E2 -8169.865} C_VEL
LIN {X 0,Y 458.56,Z 509.187,A -85,B 0,C 180,E1 -8170.76,E2 -8170.76} C_VEL
LIN {X 0,Y 457.604,Z 521.667,A -85,B 0,C 180,E1 -8171.764,E2 -8171.764} C_VEL
LIN {X 0,Y 456.651,Z 534.295,A -85,B 0,C 180,E1 -8172.997,E2 -8172.997} C_VEL
LIN {X 0,Y 455.754,Z 545.738,A -85,B 0,C 180,E1 -8174.344,E2 -8174.344} C_VEL
LIN {X 0,Y 454.964,Z 555.364,A -85,B 0,C 180,E1 -8175.69,E2 -8175.69} C_VEL
LIN {X 0,Y 454.164,Z 564.998,A -85,B 0,C 180,E1 -8177.298,E2 -8177.298} C_VEL
LIN {X 0,Y 453.658,Z 572.64,A -85,B 0,C 180,E1 -8178.834,E2 -8178.834} C_VEL
LIN {X 0,Y 453.17,Z 579.962,A -85,B 0,C 180,E1 -8180.628,E2 -8180.628} C_VEL
LIN {X 0,Y 452.859,Z 585.77,A -85,B 0,C 180,E1 -8182.419,E2 -8182.419} C_VEL
LIN {X 0,Y 452.763,Z 589.205,A -85,B 0,C 180,E1 -8183.762,E2 -8183.762} C_VEL
LIN {X 0,Y 452.542,Z 592.693,A -85,B 0,C 180,E1 -8185.546,E2 -8185.546} C_VEL
LIN {X 0,Y 452.544,Z 594.996,A -85,B 0,C 180,E1 -8187.329,E2 -8187.329} C_VEL
LIN {X 0,Y 452.456,Z 596.178,A -85,B 0,C 180,E1 -8189.11,E2 -8189.11} C_VEL
LIN {X 0,Y 452.457,Z 596.195,A -85,B 0,C 180,E1 -8190.89,E2 -8190.89} C_VEL
LIN {X 0,Y 452.545,Z 595.082,A -85,B 0,C 180,E1 -8192.67,E2 -8192.67} C_VEL
LIN {X 0,Y 452.54,Z 592.846,A -85,B 0,C 180,E1 -8194.453,E2 -8194.453} C_VEL
LIN {X 0,Y 452.752,Z 589.421,A -85,B 0,C 180,E1 -8196.238,E2 -8196.238} C_VEL
LIN {X 0,Y 452.93,Z 584.737,A -85,B 0,C 180,E1 -8198.027,E2 -8198.027} C_VEL
LIN {X 0,Y 453.262,Z 578.664,A -85,B 0,C 180,E1 -8199.82,E2 -8199.82} C_VEL
LIN {X 0,Y 453.864,Z 571.008,A -85,B 0,C 180,E1 -8201.613,E2 -8201.613} C_VEL
LIN {X 0,Y 454.321,Z 563.113,A -85,B 0,C 180,E1 -8203.141,E2 -8203.141} C_VEL
LIN {X 0,Y 455.189,Z 553.01,A -85,B 0,C 180,E1 -8204.759,E2 -8204.759} C_VEL
LIN {X 0,Y 455.981,Z 542.919,A -85,B 0,C 180,E1 -8206.107,E2 -8206.107} C_VEL
LIN {X 0,Y 456.877,Z 531.985,A -85,B 0,C 180,E1 -8207.337,E2 -8207.337} C_VEL
LIN {X 0,Y 457.721,Z 520.128,A -85,B 0,C 180,E1 -8208.462,E2 -8208.462} C_VEL
LIN {X 0,Y 458.726,Z 507.31,A -85,B 0,C 180,E1 -8209.464,E2 -8209.464} C_VEL
LIN {X 0,Y 459.442,Z 495.231,A -85,B 0,C 180,E1 -8210.248,E2 -8210.248} C_VEL
LIN {X 0,Y 460.219,Z 481.066,A -85,B 0,C 180,E1 -8210.979,E2 -8210.979} C_VEL
LIN {X 0,Y 460.808,Z 466.473,A -85,B 0,C 180,E1 -8211.55,E2 -8211.55} C_VEL
LIN {X 0,Y 461.2,Z 451.879,A -85,B 0,C 180,E1 -8211.951,E2 -8211.951} C_VEL
LIN {X 0,Y 462.762,Z 340.849,A -85,B 0,C 180,E1 -8213.731,E2 -8213.731} C_VEL
LIN {X 0,Y 462.99,Z 307.826,A -85,B 0,C 180,E1 -8214.268,E2 -8214.268} C_VEL
LIN {X 0,Y 460.572,Z 298.429,A -85,B 0,C 180,E1 -8214.564,E2 -8214.564} C_VEL
LIN {X 0,Y 455.866,Z 287.079,A -85,B 0,C 180,E1 -8215.038,E2 -8215.038} C_VEL
LIN {X 0,Y 453.469,Z 276.627,A -85,B 0,C 180,E1 -8217.144,E2 -8217.144} C_VEL
LIN {X 0,Y 453.468,Z 276.627,A -85,B 0,C 180,E1 -8219.783,E2 -8219.783} C_VEL
LIN {X 0,Y 453.463,Z 276.626,A -85,B 0,C 180,E1 -8223.184,E2 -8223.184} C_VEL
LIN {X 0,Y 453.439,Z 276.624,A -85,B 0,C 180,E1 -8226.296,E2 -8226.296} C_VEL
LIN {X 0,Y 453.44,Z 276.627,A -85,B 0,C 180,E1 -8229.455,E2 -8229.455} C_VEL
LIN {X 0,Y 453.433,Z 276.625,A -85,B 0,C 180,E1 -8231.929,E2 -8231.929} C_VEL
LIN {X 0,Y 453.473,Z 276.621,A -85,B 0,C 180,E1 -8235.472,E2 -8235.472} C_VEL
LIN {X 0,Y 453.461,Z 276.621,A -85,B 0,C 180,E1 -8239.387,E2 -8239.387} C_VEL
LIN {X 0,Y 453.429,Z 276.616,A -85,B 0,C 180,E1 -8242.808,E2 -8242.808} C_VEL
LIN {X 0,Y 453.451,Z 276.622,A -85,B 0,C 180,E1 -8246.085,E2 -8246.085} C_VEL
LIN {X 0,Y 453.444,Z 276.623,A -85,B 0,C 180,E1 -8249.238,E2 -8249.238} C_VEL
LIN {X 0,Y 453.468,Z 276.623,A -85,B 0,C 180,E1 -8252.293,E2 -8252.293} C_VEL
LIN {X 0,Y 453.463,Z 276.621,A -85,B 0,C 180,E1 -8255.263,E2 -8255.263} C_VEL
LIN {X 0,Y 453.474,Z 276.625,A -85,B 0,C 180,E1 -8258.417,E2 -8258.417} C_VEL
LIN {X 0,Y 453.483,Z 276.615,A -85,B 0,C 180,E1 -8261.007,E2 -8261.007} C_VEL
LIN {X 0,Y 453.515,Z 276.614,A -85,B 0,C 180,E1 -8264.725,E2 -8264.725} C_VEL
LIN {X 0,Y 453.555,Z 276.617,A -85,B 0,C 180,E1 -8268.379,E2 -8268.379} C_VEL
LIN {X 0,Y 453.559,Z 276.604,A -85,B 0,C 180,E1 -8271.086,E2 -8271.086} C_VEL
LIN {X 0,Y 453.627,Z 276.603,A -85,B 0,C 180,E1 -8273.774,E2 -8273.774} C_VEL
LIN {X 0,Y 453.73,Z 276.586,A -85,B 0,C 180,E1 -8277.337,E2 -8277.337} C_VEL
LIN {X 0,Y 453.766,Z 276.587,A -85,B 0,C 180,E1 -8280,E2 -8280} C_VEL
LIN {X 0,Y 453.71,Z 276.592,A -85,B 0,C 180,E1 -8282.663,E2 -8282.663} C_VEL
LIN {X 0,Y 453.641,Z 276.599,A -85,B 0,C 180,E1 -8286.226,E2 -8286.226} C_VEL
LIN {X 0,Y 453.58,Z 276.606,A -85,B 0,C 180,E1 -8288.914,E2 -8288.914} C_VEL
LIN {X 0,Y 453.562,Z 276.611,A -85,B 0,C 180,E1 -8292.529,E2 -8292.529} C_VEL
LIN {X 0,Y 453.543,Z 276.616,A -85,B 0,C 180,E1 -8296.196,E2 -8296.196} C_VEL
LIN {X 0,Y 453.515,Z 276.612,A -85,B 0,C 180,E1 -8299.039,E2 -8299.039} C_VEL
LIN {X 0,Y 453.475,Z 276.627,A -85,B 0,C 180,E1 -8301.836,E2 -8301.836} C_VEL
LIN {X 0,Y 453.498,Z 276.602,A -85,B 0,C 180,E1 -8304.735,E2 -8304.735} C_VEL
LIN {X 0,Y 453.504,Z 276.621,A -85,B 0,C 180,E1 -8307.953,E2 -8307.953} C_VEL
LIN {X 0,Y 453.473,Z 276.614,A -85,B 0,C 180,E1 -8310.76,E2 -8310.76} C_VEL
LIN {X 0,Y 453.476,Z 276.623,A -85,B 0,C 180,E1 -8313.913,E2 -8313.913} C_VEL
LIN {X 0,Y 453.451,Z 276.618,A -85,B 0,C 180,E1 -8317.19,E2 -8317.19} C_VEL
LIN {X 0,Y 453.515,Z 276.617,A -85,B 0,C 180,E1 -8319.447,E2 -8319.447} C_VEL
LIN {X 0,Y 453.461,Z 276.623,A -85,B 0,C 180,E1 -8322.995,E2 -8322.995} C_VEL
LIN {X 0,Y 453.462,Z 276.626,A -85,B 0,C 180,E1 -8325.779,E2 -8325.779} C_VEL
LIN {X 0,Y 453.477,Z 276.618,A -85,B 0,C 180,E1 -8328.209,E2 -8328.209} C_VEL
LIN {X 0,Y 453.493,Z 276.619,A -85,B 0,C 180,E1 -8330.794,E2 -8330.794} C_VEL
LIN {X 0,Y 453.455,Z 276.628,A -85,B 0,C 180,E1 -8333.918,E2 -8333.918} C_VEL
LIN {X 0,Y 453.482,Z 276.625,A -85,B 0,C 180,E1 -8337.152,E2 -8337.152} C_VEL
LIN {X 0,Y 453.497,Z 276.83,A -85,B 0,C 180,E1 -8338.468,E2 -8338.468} C_VEL
LIN {X 0,Y 457.031,Z 290.794,A -85,B 0,C 180,E1 -8340.922,E2 -8340.922} C_VEL
LIN {X 0,Y 458.67,Z 297.99,A -85,B 0,C 180,E1 -8342.139,E2 -8342.139} C_VEL
LIN {X 0,Y 458.311,Z 306.172,A -85,B 0,C 180,E1 -8343.373,E2 -8343.373} C_VEL
LIN {X 0,Y 457.62,Z 317.737,A -85,B 0,C 180,E1 -8345.097,E2 -8345.097} C_VEL
LIN {X 0,Y 462.857,Z 345.858,A -85,B 0,C 180,E1 -8345.867,E2 -8345.867} C_VEL
LIN {X 0,Y 460.98,Z 483.693,A -85,B 0,C 180,E1 -8348.067,E2 -8348.067} C_VEL
LIN {X 0,Y 460.42,Z 499.265,A -85,B 0,C 180,E1 -8348.481,E2 -8348.481} C_VEL
LIN {X 0,Y 459.687,Z 514.86,A -85,B 0,C 180,E1 -8349.089,E2 -8349.089} C_VEL
LIN {X 0,Y 458.779,Z 529.279,A -85,B 0,C 180,E1 -8349.838,E2 -8349.838} C_VEL
LIN {X 0,Y 457.85,Z 542.802,A -85,B 0,C 180,E1 -8350.73,E2 -8350.73} C_VEL
LIN {X 0,Y 456.797,Z 556.575,A -85,B 0,C 180,E1 -8351.847,E2 -8351.847} C_VEL
LIN {X 0,Y 455.752,Z 569.072,A -85,B 0,C 180,E1 -8353.081,E2 -8353.081} C_VEL
LIN {X 0,Y 455.014,Z 579.513,A -85,B 0,C 180,E1 -8354.318,E2 -8354.318} C_VEL
LIN {X 0,Y 454.333,Z 589.234,A -85,B 0,C 180,E1 -8355.671,E2 -8355.671} C_VEL
LIN {X 0,Y 453.627,Z 598.783,A -85,B 0,C 180,E1 -8357.246,E2 -8357.246} C_VEL
LIN {X 0,Y 453.281,Z 606.75,A -85,B 0,C 180,E1 -8358.825,E2 -8358.825} C_VEL
LIN {X 0,Y 452.814,Z 614.183,A -85,B 0,C 180,E1 -8360.621,E2 -8360.621} C_VEL
LIN {X 0,Y 452.646,Z 620.088,A -85,B 0,C 180,E1 -8362.417,E2 -8362.417} C_VEL
LIN {X 0,Y 452.542,Z 623.597,A -85,B 0,C 180,E1 -8363.759,E2 -8363.759} C_VEL
LIN {X 0,Y 452.45,Z 627.144,A -85,B 0,C 180,E1 -8365.546,E2 -8365.546} C_VEL
LIN {X 0,Y 452.501,Z 629.482,A -85,B 0,C 180,E1 -8367.33,E2 -8367.33} C_VEL
LIN {X 0,Y 452.454,Z 630.655,A -85,B 0,C 180,E1 -8369.11,E2 -8369.11} C_VEL
LIN {X 0,Y 452.454,Z 630.654,A -85,B 0,C 180,E1 -8370.89,E2 -8370.89} C_VEL
LIN {X 0,Y 452.501,Z 629.476,A -85,B 0,C 180,E1 -8372.671,E2 -8372.671} C_VEL
LIN {X 0,Y 452.45,Z 627.137,A -85,B 0,C 180,E1 -8374.455,E2 -8374.455} C_VEL
LIN {X 0,Y 452.513,Z 623.484,A -85,B 0,C 180,E1 -8376.287,E2 -8376.287} C_VEL
LIN {X 0,Y 452.671,Z 618.753,A -85,B 0,C 180,E1 -8378.033,E2 -8378.033} C_VEL
LIN {X 0,Y 452.87,Z 612.485,A -85,B 0,C 180,E1 -8379.829,E2 -8379.829} C_VEL
LIN {X 0,Y 453.291,Z 605.714,A -85,B 0,C 180,E1 -8381.402,E2 -8381.402} C_VEL
LIN {X 0,Y 453.761,Z 597.527,A -85,B 0,C 180,E1 -8382.979,E2 -8382.979} C_VEL
LIN {X 0,Y 454.437,Z 587.72,A -85,B 0,C 180,E1 -8384.556,E2 -8384.556} C_VEL
LIN {X 0,Y 455.184,Z 577.698,A -85,B 0,C 180,E1 -8385.906,E2 -8385.906} C_VEL
LIN {X 0,Y 456.022,Z 566.767,A -85,B 0,C 180,E1 -8387.155,E2 -8387.155} C_VEL
LIN {X 0,Y 456.987,Z 553.953,A -85,B 0,C 180,E1 -8388.378,E2 -8388.378} C_VEL
LIN {X 0,Y 457.967,Z 541.165,A -85,B 0,C 180,E1 -8389.382,E2 -8389.382} C_VEL
LIN {X 0,Y 458.917,Z 527.221,A -85,B 0,C 180,E1 -8390.273,E2 -8390.273} C_VEL
LIN {X 0,Y 459.734,Z 513.621,A -85,B 0,C 180,E1 -8390.963,E2 -8390.963} C_VEL
LIN {X 0,Y 460.389,Z 499.168,A -85,B 0,C 180,E1 -8391.522,E2 -8391.522} C_VEL
LIN {X 0,Y 460.99,Z 483.506,A -85,B 0,C 180,E1 -8391.933,E2 -8391.933} C_VEL
LIN {X 0,Y 462.809,Z 346.577,A -85,B 0,C 180,E1 -8394.12,E2 -8394.12} C_VEL
LIN {X 0,Y 462.223,Z 342.081,A -85,B 0,C 180,E1 -8394.227,E2 -8394.227} C_VEL
LIN {X 0,Y 457.6,Z 317.666,A -85,B 0,C 180,E1 -8394.911,E2 -8394.911} C_VEL
LIN {X 0,Y 458.761,Z 299.565,A -85,B 0,C 180,E1 -8397.608,E2 -8397.608} C_VEL
LIN {X 0,Y 457.62,Z 293.362,A -85,B 0,C 180,E1 -8398.635,E2 -8398.635} C_VEL
LIN {X 0,Y 454.749,Z 281.641,A -85,B 0,C 180,E1 -8400.665,E2 -8400.665} C_VEL
LIN {X 0,Y 453.479,Z 276.621,A -85,B 0,C 180,E1 -8401.578,E2 -8401.578} C_VEL
LIN {X 0,Y 453.49,Z 276.623,A -85,B 0,C 180,E1 -8404.778,E2 -8404.778} C_VEL
LIN {X 0,Y 453.462,Z 276.627,A -85,B 0,C 180,E1 -8408.313,E2 -8408.313} C_VEL
LIN {X 0,Y 453.496,Z 276.621,A -85,B 0,C 180,E1 -8410.609,E2 -8410.609} C_VEL
LIN {X 0,Y 453.463,Z 276.626,A -85,B 0,C 180,E1 -8414.222,E2 -8414.222} C_VEL
LIN {X 0,Y 453.465,Z 276.62,A -85,B 0,C 180,E1 -8417.005,E2 -8417.005} C_VEL
LIN {X 0,Y 453.497,Z 276.617,A -85,B 0,C 180,E1 -8419.409,E2 -8419.409} C_VEL
LIN {X 0,Y 453.449,Z 276.626,A -85,B 0,C 180,E1 -8422.228,E2 -8422.228} C_VEL
LIN {X 0,Y 453.49,Z 276.615,A -85,B 0,C 180,E1 -8425.223,E2 -8425.223} C_VEL
LIN {X 0,Y 453.47,Z 276.623,A -85,B 0,C 180,E1 -8428.475,E2 -8428.475} C_VEL
LIN {X 0,Y 453.496,Z 276.614,A -85,B 0,C 180,E1 -8431.287,E2 -8431.287} C_VEL
LIN {X 0,Y 453.508,Z 276.618,A -85,B 0,C 180,E1 -8434.284,E2 -8434.284} C_VEL
LIN {X 0,Y 453.483,Z 276.614,A -85,B 0,C 180,E1 -8437.204,E2 -8437.204} C_VEL
LIN {X 0,Y 453.508,Z 276.619,A -85,B 0,C 180,E1 -8440.066,E2 -8440.066} C_VEL
LIN {X 0,Y 453.502,Z 276.617,A -85,B 0,C 180,E1 -8442.876,E2 -8442.876} C_VEL
LIN {X 0,Y 453.516,Z 276.614,A -85,B 0,C 180,E1 -8445.644,E2 -8445.644} C_VEL
LIN {X 0,Y 453.563,Z 276.607,A -85,B 0,C 180,E1 -8448.379,E2 -8448.379} C_VEL
LIN {X 0,Y 453.582,Z 276.607,A -85,B 0,C 180,E1 -8451.087,E2 -8451.087} C_VEL
LIN {X 0,Y 453.642,Z 276.6,A -85,B 0,C 180,E1 -8453.774,E2 -8453.774} C_VEL
LIN {X 0,Y 453.709,Z 276.589,A -85,B 0,C 180,E1 -8457.337,E2 -8457.337} C_VEL
LIN {X 0,Y 453.772,Z 276.587,A -85,B 0,C 180,E1 -8460,E2 -8460} C_VEL
LIN {X 0,Y 453.719,Z 276.588,A -85,B 0,C 180,E1 -8462.664,E2 -8462.664} C_VEL
LIN {X 0,Y 453.634,Z 276.599,A -85,B 0,C 180,E1 -8466.226,E2 -8466.226} C_VEL
LIN {X 0,Y 453.565,Z 276.609,A -85,B 0,C 180,E1 -8468.914,E2 -8468.914} C_VEL
LIN {X 0,Y 453.569,Z 276.608,A -85,B 0,C 180,E1 -8472.529,E2 -8472.529} C_VEL
LIN {X 0,Y 453.501,Z 276.618,A -85,B 0,C 180,E1 -8476.198,E2 -8476.198} C_VEL
LIN {X 0,Y 453.49,Z 276.616,A -85,B 0,C 180,E1 -8479.027,E2 -8479.027} C_VEL
LIN {X 0,Y 453.473,Z 276.621,A -85,B 0,C 180,E1 -8481.836,E2 -8481.836} C_VEL
LIN {X 0,Y 453.465,Z 276.621,A -85,B 0,C 180,E1 -8484.737,E2 -8484.737} C_VEL
LIN {X 0,Y 453.459,Z 276.61,A -85,B 0,C 180,E1 -8487.941,E2 -8487.941} C_VEL
LIN {X 0,Y 453.45,Z 276.623,A -85,B 0,C 180,E1 -8490.762,E2 -8490.762} C_VEL
LIN {X 0,Y 453.456,Z 276.624,A -85,B 0,C 180,E1 -8493.915,E2 -8493.915} C_VEL
LIN {X 0,Y 453.434,Z 276.628,A -85,B 0,C 180,E1 -8497.192,E2 -8497.192} C_VEL
LIN {X 0,Y 453.467,Z 276.621,A -85,B 0,C 180,E1 -8500.612,E2 -8500.612} C_VEL
LIN {X 0,Y 453.436,Z 276.623,A -85,B 0,C 180,E1 -8504.225,E2 -8504.225} C_VEL
LIN {X 0,Y 453.398,Z 276.632,A -85,B 0,C 180,E1 -8506.997,E2 -8506.997} C_VEL
LIN {X 0,Y 453.466,Z 276.626,A -85,B 0,C 180,E1 -8509.413,E2 -8509.413} C_VEL
LIN {X 0,Y 453.433,Z 276.624,A -85,B 0,C 180,E1 -8512.808,E2 -8512.808} C_VEL
LIN {X 0,Y 453.455,Z 276.621,A -85,B 0,C 180,E1 -8516.085,E2 -8516.085} C_VEL
LIN {X 0,Y 453.448,Z 276.629,A -85,B 0,C 180,E1 -8519.238,E2 -8519.238} C_VEL
LIN {X 0,Y 453.47,Z 276.622,A -85,B 0,C 180,E1 -8522.293,E2 -8522.293} C_VEL
LIN {X 0,Y 453.482,Z 276.749,A -85,B 0,C 180,E1 -8522.981,E2 -8522.981} C_VEL
LIN {X 0,Y 455.938,Z 287.319,A -85,B 0,C 180,E1 -8525.072,E2 -8525.072} C_VEL
LIN {X 0,Y 461.139,Z 300.144,A -85,B 0,C 180,E1 -8525.592,E2 -8525.592} C_VEL
LIN {X 0,Y 463.12,Z 309.434,A -85,B 0,C 180,E1 -8525.859,E2 -8525.859} C_VEL
LIN {X 0,Y 462.062,Z 397.262,A -85,B 0,C 180,E1 -8527.261,E2 -8527.261} C_VEL
LIN {X 0,Y 461.322,Z 403.108,A -85,B 0,C 180,E1 -8527.319,E2 -8527.319} C_VEL
LIN {X 0,Y 455.681,Z 422.123,A -85,B 0,C 180,E1 -8527.337,E2 -8527.337} C_VEL
LIN {X 0,Y 455.028,Z 427.964,A -85,B 0,C 180,E1 -8527.4,E2 -8527.4} C_VEL
LIN {X 0,Y 454.641,Z 453.452,A -85,B 0,C 180,E1 -8527.843,E2 -8527.843} C_VEL
LIN {X 0,Y 454.163,Z 467.962,A -85,B 0,C 180,E1 -8528.255,E2 -8528.255} C_VEL
LIN {X 0,Y 453.529,Z 482.316,A -85,B 0,C 180,E1 -8528.835,E2 -8528.835} C_VEL
LIN {X 0,Y 452.749,Z 495.89,A -85,B 0,C 180,E1 -8529.557,E2 -8529.557} C_VEL
LIN {X 0,Y 451.876,Z 509.463,A -85,B 0,C 180,E1 -8530.464,E2 -8530.464} C_VEL
LIN {X 0,Y 450.86,Z 521.943,A -85,B 0,C 180,E1 -8531.481,E2 -8531.481} C_VEL
LIN {X 0,Y 449.969,Z 533.169,A -85,B 0,C 180,E1 -8532.582,E2 -8532.582} C_VEL
LIN {X 0,Y 449.057,Z 544.244,A -85,B 0,C 180,E1 -8533.871,E2 -8533.871} C_VEL
LIN {X 0,Y 448.204,Z 554.165,A -85,B 0,C 180,E1 -8535.237,E2 -8535.237} C_VEL
LIN {X 0,Y 447.412,Z 563.552,A -85,B 0,C 180,E1 -8536.778,E2 -8536.778} C_VEL
LIN {X 0,Y 446.818,Z 571.912,A -85,B 0,C 180,E1 -8538.431,E2 -8538.431} C_VEL
LIN {X 0,Y 446.276,Z 578.565,A -85,B 0,C 180,E1 -8540.024,E2 -8540.024} C_VEL
LIN {X 0,Y 445.881,Z 584.724,A -85,B 0,C 180,E1 -8541.844,E2 -8541.844} C_VEL
LIN {X 0,Y 445.675,Z 589.478,A -85,B 0,C 180,E1 -8543.662,E2 -8543.662} C_VEL
LIN {X 0,Y 445.462,Z 592.964,A -85,B 0,C 180,E1 -8545.475,E2 -8545.475} C_VEL
LIN {X 0,Y 445.471,Z 595.266,A -85,B 0,C 180,E1 -8547.287,E2 -8547.287} C_VEL
LIN {X 0,Y 445.365,Z 596.448,A -85,B 0,C 180,E1 -8549.095,E2 -8549.095} C_VEL
LIN {X 0,Y 445.366,Z 596.465,A -85,B 0,C 180,E1 -8550.904,E2 -8550.904} C_VEL
LIN {X 0,Y 445.472,Z 595.351,A -85,B 0,C 180,E1 -8552.712,E2 -8552.712} C_VEL
LIN {X 0,Y 445.46,Z 593.116,A -85,B 0,C 180,E1 -8554.524,E2 -8554.524} C_VEL
LIN {X 0,Y 445.665,Z 589.692,A -85,B 0,C 180,E1 -8556.337,E2 -8556.337} C_VEL
LIN {X 0,Y 445.877,Z 585.007,A -85,B 0,C 180,E1 -8558.155,E2 -8558.155} C_VEL
LIN {X 0,Y 446.251,Z 578.933,A -85,B 0,C 180,E1 -8559.976,E2 -8559.976} C_VEL
LIN {X 0,Y 446.87,Z 571.278,A -85,B 0,C 180,E1 -8561.797,E2 -8561.797} C_VEL
LIN {X 0,Y 447.403,Z 563.148,A -85,B 0,C 180,E1 -8563.391,E2 -8563.391} C_VEL
LIN {X 0,Y 448.287,Z 553.279,A -85,B 0,C 180,E1 -8564.991,E2 -8564.991} C_VEL
LIN {X 0,Y 449.13,Z 543.188,A -85,B 0,C 180,E1 -8566.359,E2 -8566.359} C_VEL
LIN {X 0,Y 450.054,Z 532.725,A -85,B 0,C 180,E1 -8567.556,E2 -8567.556} C_VEL
LIN {X 0,Y 450.98,Z 520.394,A -85,B 0,C 180,E1 -8568.748,E2 -8568.748} C_VEL
LIN {X 0,Y 452.029,Z 507.574,A -85,B 0,C 180,E1 -8569.765,E2 -8569.765} C_VEL
LIN {X 0,Y 452.916,Z 493.513,A -85,B 0,C 180,E1 -8570.672,E2 -8570.672} C_VEL
LIN {X 0,Y 453.735,Z 478.948,A -85,B 0,C 180,E1 -8571.402,E2 -8571.402} C_VEL
LIN {X 0,Y 454.319,Z 463.711,A -85,B 0,C 180,E1 -8571.972,E2 -8571.972} C_VEL
LIN {X 0,Y 454.752,Z 449.146,A -85,B 0,C 180,E1 -8572.339,E2 -8572.339} C_VEL
LIN {X 0,Y 456.638,Z 316.547,A -85,B 0,C 180,E1 -8574.484,E2 -8574.484} C_VEL
LIN {X 0,Y 456.565,Z 309.285,A -85,B 0,C 180,E1 -8574.612,E2 -8574.612} C_VEL
LIN {X 0,Y 454.536,Z 301.304,A -85,B 0,C 180,E1 -8574.867,E2 -8574.867} C_VEL
LIN {X 0,Y 448.721,Z 287.31,A -85,B 0,C 180,E1 -8575.475,E2 -8575.475} C_VEL
LIN {X 0,Y 446.43,Z 277.503,A -85,B 0,C 180,E1 -8577.513,E2 -8577.513} C_VEL
LIN {X 0,Y 446.417,Z 277.506,A -85,B 0,C 180,E1 -8580.25,E2 -8580.25} C_VEL
LIN {X 0,Y 446.423,Z 277.503,A -85,B 0,C 180,E1 -8583.449,E2 -8583.449} C_VEL
LIN {X 0,Y 446.391,Z 277.505,A -85,B 0,C 180,E1 -8586.746,E2 -8586.746} C_VEL
LIN {X 0,Y 446.395,Z 277.504,A -85,B 0,C 180,E1 -8590.203,E2 -8590.203} C_VEL
LIN {X 0,Y 446.378,Z 277.5,A -85,B 0,C 180,E1 -8593.594,E2 -8593.594} C_VEL
LIN {X 0,Y 446.376,Z 277.508,A -85,B 0,C 180,E1 -8596.406,E2 -8596.406} C_VEL
LIN {X 0,Y 446.384,Z 277.502,A -85,B 0,C 180,E1 -8599.796,E2 -8599.796} C_VEL
LIN {X 0,Y 446.387,Z 277.488,A -85,B 0,C 180,E1 -8603.253,E2 -8603.253} C_VEL
LIN {X 0,Y 446.422,Z 277.503,A -85,B 0,C 180,E1 -8606.55,E2 -8606.55} C_VEL
LIN {X 0,Y 446.411,Z 277.5,A -85,B 0,C 180,E1 -8609.983,E2 -8609.983} C_VEL
LIN {X 0,Y 446.389,Z 277.504,A -85,B 0,C 180,E1 -8612.833,E2 -8612.833} C_VEL
LIN {X 0,Y 446.416,Z 277.5,A -85,B 0,C 180,E1 -8615.937,E2 -8615.937} C_VEL
LIN {X 0,Y 446.439,Z 277.5,A -85,B 0,C 180,E1 -8618.772,E2 -8618.772} C_VEL
LIN {X 0,Y 446.412,Z 277.494,A -85,B 0,C 180,E1 -8621.647,E2 -8621.647} C_VEL
LIN {X 0,Y 446.455,Z 277.497,A -85,B 0,C 180,E1 -8624.478,E2 -8624.478} C_VEL
LIN {X 0,Y 446.515,Z 277.486,A -85,B 0,C 180,E1 -8627.384,E2 -8627.384} C_VEL
LIN {X 0,Y 446.51,Z 277.483,A -85,B 0,C 180,E1 -8630.944,E2 -8630.944} C_VEL
LIN {X 0,Y 446.598,Z 277.478,A -85,B 0,C 180,E1 -8633.676,E2 -8633.676} C_VEL
LIN {X 0,Y 446.677,Z 277.465,A -85,B 0,C 180,E1 -8637.294,E2 -8637.294} C_VEL
LIN {X 0,Y 446.716,Z 277.465,A -85,B 0,C 180,E1 -8640,E2 -8640} C_VEL
LIN {X 0,Y 446.659,Z 277.47,A -85,B 0,C 180,E1 -8642.705,E2 -8642.705} C_VEL
LIN {X 0,Y 446.61,Z 277.475,A -85,B 0,C 180,E1 -8646.324,E2 -8646.324} C_VEL
LIN {X 0,Y 446.528,Z 277.484,A -85,B 0,C 180,E1 -8649.055,E2 -8649.055} C_VEL
LIN {X 0,Y 446.52,Z 277.487,A -85,B 0,C 180,E1 -8652.73,E2 -8652.73} C_VEL
LIN {X 0,Y 446.494,Z 277.495,A -85,B 0,C 180,E1 -8656.227,E2 -8656.227} C_VEL
LIN {X 0,Y 446.467,Z 277.491,A -85,B 0,C 180,E1 -8659.303,E2 -8659.303} C_VEL
LIN {X 0,Y 446.416,Z 277.501,A -85,B 0,C 180,E1 -8662.2,E2 -8662.2} C_VEL
LIN {X 0,Y 446.441,Z 277.481,A -85,B 0,C 180,E1 -8665.153,E2 -8665.153} C_VEL
LIN {X 0,Y 446.447,Z 277.499,A -85,B 0,C 180,E1 -8668.181,E2 -8668.181} C_VEL
LIN {X 0,Y 446.414,Z 277.493,A -85,B 0,C 180,E1 -8671.3,E2 -8671.3} C_VEL
LIN {X 0,Y 446.428,Z 277.498,A -85,B 0,C 180,E1 -8674.523,E2 -8674.523} C_VEL
LIN {X 0,Y 446.414,Z 277.496,A -85,B 0,C 180,E1 -8678.079,E2 -8678.079} C_VEL
LIN {X 0,Y 446.425,Z 277.498,A -85,B 0,C 180,E1 -8680.918,E2 -8680.918} C_VEL
LIN {X 0,Y 446.398,Z 277.506,A -85,B 0,C 180,E1 -8683.846,E2 -8683.846} C_VEL
LIN {X 0,Y 446.396,Z 277.501,A -85,B 0,C 180,E1 -8686.404,E2 -8686.404} C_VEL
LIN {X 0,Y 446.425,Z 277.496,A -85,B 0,C 180,E1 -8689.083,E2 -8689.083} C_VEL
LIN {X 0,Y 446.408,Z 277.502,A -85,B 0,C 180,E1 -8692.122,E2 -8692.122} C_VEL
LIN {X 0,Y 446.429,Z 277.503,A -85,B 0,C 180,E1 -8695.477,E2 -8695.477} C_VEL
LIN {X 0,Y 446.452,Z 277.694,A -85,B 0,C 180,E1 -8698.1,E2 -8698.1} C_VEL
LIN {X 0,Y 450.291,Z 292.821,A -85,B 0,C 180,E1 -8700.809,E2 -8700.809} C_VEL
LIN {X 0,Y 451.94,Z 300.943,A -85,B 0,C 180,E1 -8702.192,E2 -8702.192} C_VEL
LIN {X 0,Y 450.911,Z 317.473,A -85,B 0,C 180,E1 -8704.702,E2 -8704.702} C_VEL
LIN {X 0,Y 456.361,Z 346.788,A -85,B 0,C 180,E1 -8705.521,E2 -8705.521} C_VEL
LIN {X 0,Y 454.415,Z 483.438,A -85,B 0,C 180,E1 -8707.734,E2 -8707.734} C_VEL
LIN {X 0,Y 453.808,Z 499.003,A -85,B 0,C 180,E1 -8708.151,E2 -8708.151} C_VEL
LIN {X 0,Y 453.042,Z 514.317,A -85,B 0,C 180,E1 -8708.755,E2 -8708.755} C_VEL
LIN {X 0,Y 452.087,Z 529.012,A -85,B 0,C 180,E1 -8709.527,E2 -8709.527} C_VEL
LIN {X 0,Y 451.13,Z 542.535,A -85,B 0,C 180,E1 -8710.431,E2 -8710.431} C_VEL
LIN {X 0,Y 449.984,Z 556.305,A -85,B 0,C 180,E1 -8711.563,E2 -8711.563} C_VEL
LIN {X 0,Y 448.972,Z 567.9,A -85,B 0,C 180,E1 -8712.72,E2 -8712.72} C_VEL
LIN {X 0,Y 448.121,Z 579.242,A -85,B 0,C 180,E1 -8714.071,E2 -8714.071} C_VEL
LIN {X 0,Y 447.375,Z 588.962,A -85,B 0,C 180,E1 -8715.443,E2 -8715.443} C_VEL
LIN {X 0,Y 446.616,Z 598.51,A -85,B 0,C 180,E1 -8717.042,E2 -8717.042} C_VEL
LIN {X 0,Y 446.232,Z 606.477,A -85,B 0,C 180,E1 -8718.646,E2 -8718.646} C_VEL
LIN {X 0,Y 445.761,Z 613.912,A -85,B 0,C 180,E1 -8720.471,E2 -8720.471} C_VEL
LIN {X 0,Y 445.551,Z 619.816,A -85,B 0,C 180,E1 -8722.295,E2 -8722.295} C_VEL
LIN {X 0,Y 445.451,Z 623.428,A -85,B 0,C 180,E1 -8723.703,E2 -8723.703} C_VEL
LIN {X 0,Y 445.371,Z 626.874,A -85,B 0,C 180,E1 -8725.475,E2 -8725.475} C_VEL
LIN {X 0,Y 445.426,Z 629.212,A -85,B 0,C 180,E1 -8727.287,E2 -8727.287} C_VEL
LIN {X 0,Y 445.363,Z 630.385,A -85,B 0,C 180,E1 -8729.096,E2 -8729.096} C_VEL
LIN {X 0,Y 445.363,Z 630.384,A -85,B 0,C 180,E1 -8730.905,E2 -8730.905} C_VEL
LIN {X 0,Y 445.426,Z 629.206,A -85,B 0,C 180,E1 -8732.714,E2 -8732.714} C_VEL
LIN {X 0,Y 445.371,Z 626.866,A -85,B 0,C 180,E1 -8734.526,E2 -8734.526} C_VEL
LIN {X 0,Y 445.43,Z 623.321,A -85,B 0,C 180,E1 -8736.341,E2 -8736.341} C_VEL
LIN {X 0,Y 445.594,Z 618.48,A -85,B 0,C 180,E1 -8738.161,E2 -8738.161} C_VEL
LIN {X 0,Y 445.814,Z 612.211,A -85,B 0,C 180,E1 -8739.987,E2 -8739.987} C_VEL
LIN {X 0,Y 446.224,Z 605.438,A -85,B 0,C 180,E1 -8741.585,E2 -8741.585} C_VEL
LIN {X 0,Y 446.734,Z 597.251,A -85,B 0,C 180,E1 -8743.187,E2 -8743.187} C_VEL
LIN {X 0,Y 447.471,Z 587.444,A -85,B 0,C 180,E1 -8744.787,E2 -8744.787} C_VEL
LIN {X 0,Y 448.29,Z 577.422,A -85,B 0,C 180,E1 -8746.158,E2 -8746.158} C_VEL
LIN {X 0,Y 449.1,Z 567.361,A -85,B 0,C 180,E1 -8747.332,E2 -8747.332} C_VEL
LIN {X 0,Y 450.092,Z 554.975,A -85,B 0,C 180,E1 -8748.551,E2 -8748.551} C_VEL
LIN {X 0,Y 451.104,Z 542.478,A -85,B 0,C 180,E1 -8749.571,E2 -8749.571} C_VEL
LIN {X 0,Y 452.105,Z 528.937,A -85,B 0,C 180,E1 -8750.473,E2 -8750.473} C_VEL
LIN {X 0,Y 453.033,Z 514.308,A -85,B 0,C 180,E1 -8751.244,E2 -8751.244} C_VEL
LIN {X 0,Y 453.767,Z 498.888,A -85,B 0,C 180,E1 -8751.852,E2 -8751.852} C_VEL
LIN {X 0,Y 454.404,Z 483.22,A -85,B 0,C 180,E1 -8752.268,E2 -8752.268} C_VEL
LIN {X 0,Y 456.314,Z 346.969,A -85,B 0,C 180,E1 -8754.475,E2 -8754.475} C_VEL
LIN {X 0,Y 452.402,Z 325.483,A -85,B 0,C 180,E1 -8755.065,E2 -8755.065} C_VEL
LIN {X 0,Y 450.85,Z 317.482,A -85,B 0,C 180,E1 -8755.295,E2 -8755.295} C_VEL
LIN {X 0,Y 451.94,Z 300.9,A -85,B 0,C 180,E1 -8757.809,E2 -8757.809} C_VEL
LIN {X 0,Y 449.531,Z 289.513,A -85,B 0,C 180,E1 -8759.761,E2 -8759.761} C_VEL
LIN {X 0,Y 446.433,Z 277.501,A -85,B 0,C 180,E1 -8761.944,E2 -8761.944} C_VEL
LIN {X 0,Y 446.431,Z 277.501,A -85,B 0,C 180,E1 -8765.054,E2 -8765.054} C_VEL
LIN {X 0,Y 446.415,Z 277.502,A -85,B 0,C 180,E1 -8768.079,E2 -8768.079} C_VEL
LIN {X 0,Y 446.425,Z 277.501,A -85,B 0,C 180,E1 -8770.917,E2 -8770.917} C_VEL
LIN {X 0,Y 446.401,Z 277.503,A -85,B 0,C 180,E1 -8773.847,E2 -8773.847} C_VEL
LIN {X 0,Y 446.399,Z 277.498,A -85,B 0,C 180,E1 -8776.404,E2 -8776.404} C_VEL
LIN {X 0,Y 446.43,Z 277.498,A -85,B 0,C 180,E1 -8779.083,E2 -8779.083} C_VEL
LIN {X 0,Y 446.409,Z 277.503,A -85,B 0,C 180,E1 -8782.121,E2 -8782.121} C_VEL
LIN {X 0,Y 446.432,Z 277.495,A -85,B 0,C 180,E1 -8785.477,E2 -8785.477} C_VEL
LIN {X 0,Y 446.42,Z 277.499,A -85,B 0,C 180,E1 -8788.7,E2 -8788.7} C_VEL
LIN {X 0,Y 446.454,Z 277.494,A -85,B 0,C 180,E1 -8791.83,E2 -8791.83} C_VEL
LIN {X 0,Y 446.443,Z 277.495,A -85,B 0,C 180,E1 -8794.847,E2 -8794.847} C_VEL
LIN {X 0,Y 446.453,Z 277.499,A -85,B 0,C 180,E1 -8798.245,E2 -8798.245} C_VEL
LIN {X 0,Y 446.455,Z 277.493,A -85,B 0,C 180,E1 -8801.649,E2 -8801.649} C_VEL
LIN {X 0,Y 446.512,Z 277.486,A -85,B 0,C 180,E1 -8804.48,E2 -8804.48} C_VEL
LIN {X 0,Y 446.522,Z 277.486,A -85,B 0,C 180,E1 -8808.193,E2 -8808.193} C_VEL
LIN {X 0,Y 446.531,Z 277.485,A -85,B 0,C 180,E1 -8810.945,E2 -8810.945} C_VEL
LIN {X 0,Y 446.611,Z 277.474,A -85,B 0,C 180,E1 -8813.676,E2 -8813.676} C_VEL
LIN {X 0,Y 446.658,Z 277.467,A -85,B 0,C 180,E1 -8817.295,E2 -8817.295} C_VEL
LIN {X 0,Y 446.722,Z 277.465,A -85,B 0,C 180,E1 -8820,E2 -8820} C_VEL
LIN {X 0,Y 446.668,Z 277.466,A -85,B 0,C 180,E1 -8822.706,E2 -8822.706} C_VEL
LIN {X 0,Y 446.604,Z 277.474,A -85,B 0,C 180,E1 -8826.324,E2 -8826.324} C_VEL
LIN {X 0,Y 446.516,Z 277.487,A -85,B 0,C 180,E1 -8829.056,E2 -8829.056} C_VEL
LIN {X 0,Y 446.526,Z 277.485,A -85,B 0,C 180,E1 -8832.73,E2 -8832.73} C_VEL
LIN {X 0,Y 446.455,Z 277.496,A -85,B 0,C 180,E1 -8836.207,E2 -8836.207} C_VEL
LIN {X 0,Y 446.436,Z 277.496,A -85,B 0,C 180,E1 -8839.305,E2 -8839.305} C_VEL
LIN {X 0,Y 446.411,Z 277.497,A -85,B 0,C 180,E1 -8842.2,E2 -8842.2} C_VEL
LIN {X 0,Y 446.416,Z 277.503,A -85,B 0,C 180,E1 -8845.155,E2 -8845.155} C_VEL
LIN {X 0,Y 446.419,Z 277.486,A -85,B 0,C 180,E1 -8848.183,E2 -8848.183} C_VEL
LIN {X 0,Y 446.392,Z 277.507,A -85,B 0,C 180,E1 -8851.302,E2 -8851.302} C_VEL
LIN {X 0,Y 446.414,Z 277.5,A -85,B 0,C 180,E1 -8854.524,E2 -8854.524} C_VEL
LIN {X 0,Y 446.389,Z 277.502,A -85,B 0,C 180,E1 -8857.881,E2 -8857.881} C_VEL
LIN {X 0,Y 446.397,Z 277.504,A -85,B 0,C 180,E1 -8861.395,E2 -8861.395} C_VEL
LIN {X 0,Y 446.404,Z 277.505,A -85,B 0,C 180,E1 -8865.11,E2 -8865.11} C_VEL
LIN {X 0,Y 446.396,Z 277.501,A -85,B 0,C 180,E1 -8868.605,E2 -8868.605} C_VEL
LIN {X 0,Y 446.387,Z 277.502,A -85,B 0,C 180,E1 -8872.118,E2 -8872.118} C_VEL
LIN {X 0,Y 446.414,Z 277.499,A -85,B 0,C 180,E1 -8875.475,E2 -8875.475} C_VEL
LIN {X 0,Y 446.39,Z 277.503,A -85,B 0,C 180,E1 -8878.697,E2 -8878.697} C_VEL
LIN {X 0,Y 446.402,Z 277.505,A -85,B 0,C 180,E1 -8881.842,E2 -8881.842} C_VEL
LIN {X 0,Y 446.451,Z 277.676,A -85,B 0,C 180,E1 -8882.647,E2 -8882.647} C_VEL
LIN {X 0,Y 448.813,Z 287.666,A -85,B 0,C 180,E1 -8884.649,E2 -8884.649} C_VEL
LIN {X 0,Y 454.826,Z 302.05,A -85,B 0,C 180,E1 -8885.258,E2 -8885.258} C_VEL
LIN {X 0,Y 456.667,Z 310.078,A -85,B 0,C 180,E1 -8885.502,E2 -8885.502} C_VEL
LIN {X 0,Y 455.194,Z 415.779,A -85,B 0,C 180,E1 -8887.204,E2 -8887.204} C_VEL
LIN {X 0,Y 455.028,Z 427.964,A -85,B 0,C 180,E1 -8887.4,E2 -8887.4} C_VEL
LIN {X 0,Y 454.372,Z 433.813,A -85,B 0,C 180,E1 -8887.461,E2 -8887.461} C_VEL
LIN {X 0,Y 448.683,Z 452.817,A -85,B 0,C 180,E1 -8887.509,E2 -8887.509} C_VEL
LIN {X 0,Y 447.922,Z 458.614,A -85,B 0,C 180,E1 -8887.623,E2 -8887.623} C_VEL
LIN {X 0,Y 447.331,Z 474.065,A -85,B 0,C 180,E1 -8888.138,E2 -8888.138} C_VEL
LIN {X 0,Y 446.662,Z 487.997,A -85,B 0,C 180,E1 -8888.783,E2 -8888.783} C_VEL
LIN {X 0,Y 445.75,Z 501.573,A -85,B 0,C 180,E1 -8889.583,E2 -8889.583} C_VEL
LIN {X 0,Y 444.674,Z 515.569,A -85,B 0,C 180,E1 -8890.615,E2 -8890.615} C_VEL
LIN {X 0,Y 443.626,Z 528.089,A -85,B 0,C 180,E1 -8891.75,E2 -8891.75} C_VEL
LIN {X 0,Y 442.688,Z 538.891,A -85,B 0,C 180,E1 -8892.92,E2 -8892.92} C_VEL
LIN {X 0,Y 441.708,Z 549.685,A -85,B 0,C 180,E1 -8894.306,E2 -8894.306} C_VEL
LIN {X 0,Y 440.882,Z 558.835,A -85,B 0,C 180,E1 -8895.695,E2 -8895.695} C_VEL
LIN {X 0,Y 440.132,Z 567.774,A -85,B 0,C 180,E1 -8897.316,E2 -8897.316} C_VEL
LIN {X 0,Y 439.481,Z 575.183,A -85,B 0,C 180,E1 -8898.936,E2 -8898.936} C_VEL
LIN {X 0,Y 439.031,Z 582.102,A -85,B 0,C 180,E1 -8900.788,E2 -8900.788} C_VEL
LIN {X 0,Y 438.688,Z 587.54,A -85,B 0,C 180,E1 -8902.636,E2 -8902.636} C_VEL
LIN {X 0,Y 438.529,Z 591.643,A -85,B 0,C 180,E1 -8904.482,E2 -8904.482} C_VEL
LIN {X 0,Y 438.403,Z 594.529,A -85,B 0,C 180,E1 -8906.323,E2 -8906.323} C_VEL
LIN {X 0,Y 438.321,Z 596.267,A -85,B 0,C 180,E1 -8908.162,E2 -8908.162} C_VEL
LIN {X 0,Y 438.278,Z 596.875,A -85,B 0,C 180,E1 -8910,E2 -8910} C_VEL
LIN {X 0,Y 438.321,Z 596.317,A -85,B 0,C 180,E1 -8911.837,E2 -8911.837} C_VEL
LIN {X 0,Y 438.403,Z 594.646,A -85,B 0,C 180,E1 -8913.676,E2 -8913.676} C_VEL
LIN {X 0,Y 438.524,Z 591.824,A -85,B 0,C 180,E1 -8915.518,E2 -8915.518} C_VEL
LIN {X 0,Y 438.683,Z 587.784,A -85,B 0,C 180,E1 -8917.363,E2 -8917.363} C_VEL
LIN {X 0,Y 439.015,Z 582.423,A -85,B 0,C 180,E1 -8919.211,E2 -8919.211} C_VEL
LIN {X 0,Y 439.46,Z 575.59,A -85,B 0,C 180,E1 -8921.064,E2 -8921.064} C_VEL
LIN {X 0,Y 440.068,Z 568.235,A -85,B 0,C 180,E1 -8922.685,E2 -8922.685} C_VEL
LIN {X 0,Y 440.856,Z 559.371,A -85,B 0,C 180,E1 -8924.305,E2 -8924.305} C_VEL
LIN {X 0,Y 441.651,Z 550.33,A -85,B 0,C 180,E1 -8925.695,E2 -8925.695} C_VEL
LIN {X 0,Y 442.598,Z 539.659,A -85,B 0,C 180,E1 -8927.083,E2 -8927.083} C_VEL
LIN {X 0,Y 443.69,Z 528.02,A -85,B 0,C 180,E1 -8928.348,E2 -8928.348} C_VEL
LIN {X 0,Y 444.738,Z 515.269,A -85,B 0,C 180,E1 -8929.501,E2 -8929.501} C_VEL
LIN {X 0,Y 445.681,Z 502.968,A -85,B 0,C 180,E1 -8930.419,E2 -8930.419} C_VEL
LIN {X 0,Y 446.513,Z 489.768,A -85,B 0,C 180,E1 -8931.224,E2 -8931.224} C_VEL
LIN {X 0,Y 447.353,Z 474.149,A -85,B 0,C 180,E1 -8931.951,E2 -8931.951} C_VEL
LIN {X 0,Y 447.928,Z 459.222,A -85,B 0,C 180,E1 -8932.454,E2 -8932.454} C_VEL
LIN {X 0,Y 448.282,Z 444.877,A -85,B 0,C 180,E1 -8932.77,E2 -8932.77} C_VEL
LIN {X 0,Y 449.967,Z 330.391,A -85,B 0,C 180,E1 -8934.637,E2 -8934.637} C_VEL
LIN {X 0,Y 450.105,Z 310.39,A -85,B 0,C 180,E1 -8934.974,E2 -8934.974} C_VEL
LIN {X 0,Y 448.303,Z 303.582,A -85,B 0,C 180,E1 -8935.201,E2 -8935.201} C_VEL
LIN {X 0,Y 441.563,Z 287.528,A -85,B 0,C 180,E1 -8935.931,E2 -8935.931} C_VEL
LIN {X 0,Y 439.391,Z 278.38,A -85,B 0,C 180,E1 -8937.866,E2 -8937.866} C_VEL
LIN {X 0,Y 439.344,Z 278.385,A -85,B 0,C 180,E1 -8940.789,E2 -8940.789} C_VEL
LIN {X 0,Y 439.353,Z 278.384,A -85,B 0,C 180,E1 -8944.046,E2 -8944.046} C_VEL
LIN {X 0,Y 439.336,Z 278.385,A -85,B 0,C 180,E1 -8946.885,E2 -8946.885} C_VEL
LIN {X 0,Y 439.344,Z 278.382,A -85,B 0,C 180,E1 -8949.84,E2 -8949.84} C_VEL
LIN {X 0,Y 439.327,Z 278.38,A -85,B 0,C 180,E1 -8952.619,E2 -8952.619} C_VEL
LIN {X 0,Y 439.37,Z 278.38,A -85,B 0,C 180,E1 -8955.267,E2 -8955.267} C_VEL
LIN {X 0,Y 439.355,Z 278.373,A -85,B 0,C 180,E1 -8958.748,E2 -8958.748} C_VEL
LIN {X 0,Y 439.348,Z 278.378,A -85,B 0,C 180,E1 -8961.612,E2 -8961.612} C_VEL
LIN {X 0,Y 439.384,Z 278.369,A -85,B 0,C 180,E1 -8964.842,E2 -8964.842} C_VEL
LIN {X 0,Y 439.343,Z 278.382,A -85,B 0,C 180,E1 -8968.137,E2 -8968.137} C_VEL
LIN {X 0,Y 439.383,Z 278.374,A -85,B 0,C 180,E1 -8971.61,E2 -8971.61} C_VEL
LIN {X 0,Y 439.363,Z 278.382,A -85,B 0,C 180,E1 -8974.412,E2 -8974.412} C_VEL
LIN {X 0,Y 439.35,Z 278.377,A -85,B 0,C 180,E1 -8977.424,E2 -8977.424} C_VEL
LIN {X 0,Y 439.384,Z 278.373,A -85,B 0,C 180,E1 -8980.684,E2 -8980.684} C_VEL
LIN {X 0,Y 439.414,Z 278.377,A -85,B 0,C 180,E1 -8984.223,E2 -8984.223} C_VEL
LIN {X 0,Y 439.483,Z 278.362,A -85,B 0,C 180,E1 -8987.285,E2 -8987.285} C_VEL
LIN {X 0,Y 439.477,Z 278.36,A -85,B 0,C 180,E1 -8990.798,E2 -8990.798} C_VEL
LIN {X 0,Y 439.552,Z 278.355,A -85,B 0,C 180,E1 -8993.574,E2 -8993.574} C_VEL
LIN {X 0,Y 439.412,Z 278.368,A -85,B 0,C 180,E1 -8995.413,E2 -8995.413} C_VEL
LIN {X 0,Y 439.63,Z 278.35,A -85,B 0,C 180,E1 -8998.168,E2 -8998.168} C_VEL
LIN {X 0,Y 439.584,Z 278.343,A -85,B 0,C 180,E1 -9000.916,E2 -9000.916} C_VEL
LIN {X 0,Y 439.61,Z 278.348,A -85,B 0,C 180,E1 -9002.749,E2 -9002.749} C_VEL
LIN {X 0,Y 439.562,Z 278.353,A -85,B 0,C 180,E1 -9006.426,E2 -9006.426} C_VEL
LIN {X 0,Y 439.492,Z 278.361,A -85,B 0,C 180,E1 -9009.202,E2 -9009.202} C_VEL
LIN {X 0,Y 439.464,Z 278.366,A -85,B 0,C 180,E1 -9012.938,E2 -9012.938} C_VEL
LIN {X 0,Y 439.445,Z 278.372,A -85,B 0,C 180,E1 -9016.348,E2 -9016.348} C_VEL
LIN {X 0,Y 439.4,Z 278.373,A -85,B 0,C 180,E1 -9019.626,E2 -9019.626} C_VEL
LIN {X 0,Y 439.362,Z 278.377,A -85,B 0,C 180,E1 -9022.575,E2 -9022.575} C_VEL
LIN {X 0,Y 439.378,Z 278.361,A -85,B 0,C 180,E1 -9025.586,E2 -9025.586} C_VEL
LIN {X 0,Y 439.398,Z 278.374,A -85,B 0,C 180,E1 -9028.675,E2 -9028.675} C_VEL
LIN {X 0,Y 439.368,Z 278.367,A -85,B 0,C 180,E1 -9032.03,E2 -9032.03} C_VEL
LIN {X 0,Y 439.393,Z 278.377,A -85,B 0,C 180,E1 -9035.341,E2 -9035.341} C_VEL
LIN {X 0,Y 439.383,Z 278.373,A -85,B 0,C 180,E1 -9038.595,E2 -9038.595} C_VEL
LIN {X 0,Y 439.387,Z 278.377,A -85,B 0,C 180,E1 -9041.257,E2 -9041.257} C_VEL
LIN {X 0,Y 439.398,Z 278.374,A -85,B 0,C 180,E1 -9044.73,E2 -9044.73} C_VEL
LIN {X 0,Y 439.394,Z 278.377,A -85,B 0,C 180,E1 -9047.796,E2 -9047.796} C_VEL
LIN {X 0,Y 439.424,Z 278.372,A -85,B 0,C 180,E1 -9050.228,E2 -9050.228} C_VEL
LIN {X 0,Y 439.373,Z 278.382,A -85,B 0,C 180,E1 -9053.713,E2 -9053.713} C_VEL
LIN {X 0,Y 439.372,Z 278.382,A -85,B 0,C 180,E1 -9057.054,E2 -9057.054} C_VEL
LIN {X 0,Y 439.422,Z 278.525,A -85,B 0,C 180,E1 -9057.712,E2 -9057.712} C_VEL
LIN {X 0,Y 443.484,Z 294.584,A -85,B 0,C 180,E1 -9060.645,E2 -9060.645} C_VEL
LIN {X 0,Y 445.093,Z 301.977,A -85,B 0,C 180,E1 -9061.934,E2 -9061.934} C_VEL
LIN {X 0,Y 444.196,Z 317.174,A -85,B 0,C 180,E1 -9064.289,E2 -9064.289} C_VEL
LIN {X 0,Y 449.858,Z 347.757,A -85,B 0,C 180,E1 -9065.164,E2 -9065.164} C_VEL
LIN {X 0,Y 447.865,Z 483.183,A -85,B 0,C 180,E1 -9067.39,E2 -9067.39} C_VEL
LIN {X 0,Y 447.22,Z 498.741,A -85,B 0,C 180,E1 -9067.812,E2 -9067.812} C_VEL
LIN {X 0,Y 446.42,Z 513.102,A -85,B 0,C 180,E1 -9068.38,E2 -9068.38} C_VEL
LIN {X 0,Y 445.546,Z 526.752,A -85,B 0,C 180,E1 -9069.091,E2 -9069.091} C_VEL
LIN {X 0,Y 444.536,Z 540.679,A -85,B 0,C 180,E1 -9070.009,E2 -9070.009} C_VEL
LIN {X 0,Y 443.401,Z 553.44,A -85,B 0,C 180,E1 -9071.039,E2 -9071.039} C_VEL
LIN {X 0,Y 442.314,Z 566.356,A -85,B 0,C 180,E1 -9072.31,E2 -9072.31} C_VEL
LIN {X 0,Y 441.556,Z 575.381,A -85,B 0,C 180,E1 -9073.352,E2 -9073.352} C_VEL
LIN {X 0,Y 440.704,Z 585.669,A -85,B 0,C 180,E1 -9074.745,E2 -9074.745} C_VEL
LIN {X 0,Y 439.84,Z 595.73,A -85,B 0,C 180,E1 -9076.368,E2 -9076.368} C_VEL
LIN {X 0,Y 439.276,Z 604.094,A -85,B 0,C 180,E1 -9077.996,E2 -9077.996} C_VEL
LIN {X 0,Y 438.924,Z 610.127,A -85,B 0,C 180,E1 -9079.39,E2 -9079.39} C_VEL
LIN {X 0,Y 438.54,Z 616.771,A -85,B 0,C 180,E1 -9081.243,E2 -9081.243} C_VEL
LIN {X 0,Y 438.394,Z 621.975,A -85,B 0,C 180,E1 -9083.095,E2 -9083.095} C_VEL
LIN {X 0,Y 438.312,Z 624.985,A -85,B 0,C 180,E1 -9084.48,E2 -9084.48} C_VEL
LIN {X 0,Y 438.264,Z 627.919,A -85,B 0,C 180,E1 -9086.323,E2 -9086.323} C_VEL
LIN {X 0,Y 438.292,Z 629.671,A -85,B 0,C 180,E1 -9088.163,E2 -9088.163} C_VEL
LIN {X 0,Y 438.277,Z 630.27,A -85,B 0,C 180,E1 -9090,E2 -9090} C_VEL
LIN {X 0,Y 438.292,Z 629.667,A -85,B 0,C 180,E1 -9091.838,E2 -9091.838} C_VEL
LIN {X 0,Y 438.264,Z 627.911,A -85,B 0,C 180,E1 -9093.678,E2 -9093.678} C_VEL
LIN {X 0,Y 438.303,Z 624.977,A -85,B 0,C 180,E1 -9095.521,E2 -9095.521} C_VEL
LIN {X 0,Y 438.407,Z 620.797,A -85,B 0,C 180,E1 -9097.369,E2 -9097.369} C_VEL
LIN {X 0,Y 438.609,Z 615.259,A -85,B 0,C 180,E1 -9099.221,E2 -9099.221} C_VEL
LIN {X 0,Y 439.072,Z 608.221,A -85,B 0,C 180,E1 -9101.075,E2 -9101.075} C_VEL
LIN {X 0,Y 439.552,Z 599.46,A -85,B 0,C 180,E1 -9102.936,E2 -9102.936} C_VEL
LIN {X 0,Y 440.297,Z 590.164,A -85,B 0,C 180,E1 -9104.561,E2 -9104.561} C_VEL
LIN {X 0,Y 441.051,Z 580.716,A -85,B 0,C 180,E1 -9105.955,E2 -9105.955} C_VEL
LIN {X 0,Y 441.972,Z 569.841,A -85,B 0,C 180,E1 -9107.306,E2 -9107.306} C_VEL
LIN {X 0,Y 443.09,Z 557.222,A -85,B 0,C 180,E1 -9108.616,E2 -9108.616} C_VEL
LIN {X 0,Y 444.264,Z 543.729,A -85,B 0,C 180,E1 -9109.764,E2 -9109.764} C_VEL
LIN {X 0,Y 445.276,Z 530.483,A -85,B 0,C 180,E1 -9110.681,E2 -9110.681} C_VEL
LIN {X 0,Y 446.245,Z 516.426,A -85,B 0,C 180,E1 -9111.457,E2 -9111.457} C_VEL
LIN {X 0,Y 447.038,Z 501.831,A -85,B 0,C 180,E1 -9112.075,E2 -9112.075} C_VEL
LIN {X 0,Y 447.694,Z 486.596,A -85,B 0,C 180,E1 -9112.529,E2 -9112.529} C_VEL
LIN {X 0,Y 448.146,Z 464.467,A -85,B 0,C 180,E1 -9112.931,E2 -9112.931} C_VEL
LIN {X 0,Y 449.823,Z 347.129,A -85,B 0,C 180,E1 -9114.844,E2 -9114.844} C_VEL
LIN {X 0,Y 444.15,Z 317.197,A -85,B 0,C 180,E1 -9115.705,E2 -9115.705} C_VEL
LIN {X 0,Y 445.139,Z 302.46,A -85,B 0,C 180,E1 -9117.98,E2 -9117.98} C_VEL
LIN {X 0,Y 442.208,Z 289.219,A -85,B 0,C 180,E1 -9120.306,E2 -9120.306} C_VEL
LIN {X 0,Y 439.379,Z 278.38,A -85,B 0,C 180,E1 -9122.323,E2 -9122.323} C_VEL
LIN {X 0,Y 439.397,Z 278.377,A -85,B 0,C 180,E1 -9125.341,E2 -9125.341} C_VEL
LIN {X 0,Y 439.372,Z 278.377,A -85,B 0,C 180,E1 -9128.597,E2 -9128.597} C_VEL
LIN {X 0,Y 439.384,Z 278.376,A -85,B 0,C 180,E1 -9131.256,E2 -9131.256} C_VEL
LIN {X 0,Y 439.401,Z 278.376,A -85,B 0,C 180,E1 -9134.73,E2 -9134.73} C_VEL
LIN {X 0,Y 439.399,Z 278.372,A -85,B 0,C 180,E1 -9137.796,E2 -9137.796} C_VEL
LIN {X 0,Y 439.397,Z 278.377,A -85,B 0,C 180,E1 -9140.224,E2 -9140.224} C_VEL
LIN {X 0,Y 439.375,Z 278.377,A -85,B 0,C 180,E1 -9143.713,E2 -9143.713} C_VEL
LIN {X 0,Y 439.376,Z 278.373,A -85,B 0,C 180,E1 -9147.054,E2 -9147.054} C_VEL
LIN {X 0,Y 439.38,Z 278.376,A -85,B 0,C 180,E1 -9150.274,E2 -9150.274} C_VEL
LIN {X 0,Y 439.384,Z 278.372,A -85,B 0,C 180,E1 -9153.393,E2 -9153.393} C_VEL
LIN {X 0,Y 439.387,Z 278.374,A -85,B 0,C 180,E1 -9156.43,E2 -9156.43} C_VEL
LIN {X 0,Y 439.392,Z 278.374,A -85,B 0,C 180,E1 -9159.397,E2 -9159.397} C_VEL
LIN {X 0,Y 439.429,Z 278.374,A -85,B 0,C 180,E1 -9162.31,E2 -9162.31} C_VEL
LIN {X 0,Y 439.452,Z 278.363,A -85,B 0,C 180,E1 -9165.174,E2 -9165.174} C_VEL
LIN {X 0,Y 439.488,Z 278.364,A -85,B 0,C 180,E1 -9168.002,E2 -9168.002} C_VEL
LIN {X 0,Y 439.506,Z 278.365,A -85,B 0,C 180,E1 -9171.726,E2 -9171.726} C_VEL
LIN {X 0,Y 439.603,Z 278.349,A -85,B 0,C 180,E1 -9174.496,E2 -9174.496} C_VEL
LIN {X 0,Y 439.631,Z 278.348,A -85,B 0,C 180,E1 -9178.168,E2 -9178.168} C_VEL
LIN {X 0,Y 439.673,Z 278.343,A -85,B 0,C 180,E1 -9180,E2 -9180} C_VEL
LIN {X 0,Y 439.62,Z 278.344,A -85,B 0,C 180,E1 -9182.749,E2 -9182.749} C_VEL
LIN {X 0,Y 439.558,Z 278.351,A -85,B 0,C 180,E1 -9186.426,E2 -9186.426} C_VEL
LIN {X 0,Y 439.483,Z 278.365,A -85,B 0,C 180,E1 -9189.202,E2 -9189.202} C_VEL
LIN {X 0,Y 439.469,Z 278.365,A -85,B 0,C 180,E1 -9192.938,E2 -9192.938} C_VEL
LIN {X 0,Y 439.402,Z 278.374,A -85,B 0,C 180,E1 -9196.326,E2 -9196.326} C_VEL
LIN {X 0,Y 439.381,Z 278.378,A -85,B 0,C 180,E1 -9199.627,E2 -9199.627} C_VEL
LIN {X 0,Y 439.356,Z 278.375,A -85,B 0,C 180,E1 -9202.576,E2 -9202.576} C_VEL
LIN {X 0,Y 439.357,Z 278.38,A -85,B 0,C 180,E1 -9205.588,E2 -9205.588} C_VEL
LIN {X 0,Y 439.38,Z 278.362,A -85,B 0,C 180,E1 -9208.676,E2 -9208.676} C_VEL
LIN {X 0,Y 439.346,Z 278.38,A -85,B 0,C 180,E1 -9212.024,E2 -9212.024} C_VEL
LIN {X 0,Y 439.385,Z 278.379,A -85,B 0,C 180,E1 -9215.337,E2 -9215.337} C_VEL
LIN {X 0,Y 439.35,Z 278.378,A -85,B 0,C 180,E1 -9218.599,E2 -9218.599} C_VEL
LIN {X 0,Y 439.347,Z 278.379,A -85,B 0,C 180,E1 -9222.21,E2 -9222.21} C_VEL
LIN {X 0,Y 439.359,Z 278.384,A -85,B 0,C 180,E1 -9225.265,E2 -9225.265} C_VEL
LIN {X 0,Y 439.349,Z 278.383,A -85,B 0,C 180,E1 -9229.015,E2 -9229.015} C_VEL
LIN {X 0,Y 439.333,Z 278.381,A -85,B 0,C 180,E1 -9232.563,E2 -9232.563} C_VEL
LIN {X 0,Y 439.388,Z 278.38,A -85,B 0,C 180,E1 -9234.842,E2 -9234.842} C_VEL
LIN {X 0,Y 439.347,Z 278.379,A -85,B 0,C 180,E1 -9238.137,E2 -9238.137} C_VEL
LIN {X 0,Y 439.378,Z 278.382,A -85,B 0,C 180,E1 -9241.323,E2 -9241.323} C_VEL
LIN {X 0,Y 439.437,Z 278.5,A -85,B 0,C 180,E1 -9242.28,E2 -9242.28} C_VEL
LIN {X 0,Y 441.56,Z 287.718,A -85,B 0,C 180,E1 -9244.197,E2 -9244.197} C_VEL
LIN {X 0,Y 448.886,Z 305.338,A -85,B 0,C 180,E1 -9244.96,E2 -9244.96} C_VEL
LIN {X 0,Y 450.218,Z 311.992,A -85,B 0,C 180,E1 -9245.155,E2 -9245.155} C_VEL
LIN {X 0,Y 448.685,Z 416.076,A -85,B 0,C 180,E1 -9246.855,E2 -9246.855} C_VEL
LIN {X 0,Y 448.092,Z 453.383,A -85,B 0,C 180,E1 -9247.493,E2 -9247.493} C_VEL
LIN {X 0,Y 447.922,Z 458.614,A -85,B 0,C 180,E1 -9247.623,E2 -9247.623} C_VEL
LIN {X 0,Y 447.173,Z 462.504,A -85,B 0,C 180,E1 -9247.695,E2 -9247.695} C_VEL
LIN {X 0,Y 441.369,Z 474.664,A -85,B 0,C 180,E1 -9247.839,E2 -9247.839} C_VEL
LIN {X 0,Y 440.597,Z 478.429,A -85,B 0,C 180,E1 -9247.971,E2 -9247.971} C_VEL
LIN {X 0,Y 439.77,Z 492.49,A -85,B 0,C 180,E1 -9248.68,E2 -9248.68} C_VEL
LIN {X 0,Y 438.889,Z 505.292,A -85,B 0,C 180,E1 -9249.495,E2 -9249.495} C_VEL
LIN {X 0,Y 437.738,Z 518.641,A -85,B 0,C 180,E1 -9250.54,E2 -9250.54} C_VEL
LIN {X 0,Y 436.65,Z 531.119,A -85,B 0,C 180,E1 -9251.736,E2 -9251.736} C_VEL
LIN {X 0,Y 435.515,Z 543.024,A -85,B 0,C 180,E1 -9253.113,E2 -9253.113} C_VEL
LIN {X 0,Y 434.567,Z 553.187,A -85,B 0,C 180,E1 -9254.523,E2 -9254.523} C_VEL
LIN {X 0,Y 433.587,Z 563.266,A -85,B 0,C 180,E1 -9256.191,E2 -9256.191} C_VEL
LIN {X 0,Y 432.921,Z 571.372,A -85,B 0,C 180,E1 -9257.816,E2 -9257.816} C_VEL
LIN {X 0,Y 432.245,Z 579.112,A -85,B 0,C 180,E1 -9259.697,E2 -9259.697} C_VEL
LIN {X 0,Y 431.791,Z 585.269,A -85,B 0,C 180,E1 -9261.576,E2 -9261.576} C_VEL
LIN {X 0,Y 431.523,Z 590.022,A -85,B 0,C 180,E1 -9263.453,E2 -9263.453} C_VEL
LIN {X 0,Y 431.317,Z 593.506,A -85,B 0,C 180,E1 -9265.326,E2 -9265.326} C_VEL
LIN {X 0,Y 431.33,Z 595.806,A -85,B 0,C 180,E1 -9267.198,E2 -9267.198} C_VEL
LIN {X 0,Y 431.193,Z 596.988,A -85,B 0,C 180,E1 -9269.066,E2 -9269.066} C_VEL
LIN {X 0,Y 431.194,Z 597.005,A -85,B 0,C 180,E1 -9270.933,E2 -9270.933} C_VEL
LIN {X 0,Y 431.33,Z 595.89,A -85,B 0,C 180,E1 -9272.801,E2 -9272.801} C_VEL
LIN {X 0,Y 431.314,Z 593.655,A -85,B 0,C 180,E1 -9274.673,E2 -9274.673} C_VEL
LIN {X 0,Y 431.522,Z 590.232,A -85,B 0,C 180,E1 -9276.546,E2 -9276.546} C_VEL
LIN {X 0,Y 431.786,Z 585.547,A -85,B 0,C 180,E1 -9278.423,E2 -9278.423} C_VEL
LIN {X 0,Y 432.21,Z 579.473,A -85,B 0,C 180,E1 -9280.303,E2 -9280.303} C_VEL
LIN {X 0,Y 432.882,Z 571.818,A -85,B 0,C 180,E1 -9282.184,E2 -9282.184} C_VEL
LIN {X 0,Y 433.537,Z 563.784,A -85,B 0,C 180,E1 -9283.81,E2 -9283.81} C_VEL
LIN {X 0,Y 434.527,Z 553.816,A -85,B 0,C 180,E1 -9285.478,E2 -9285.478} C_VEL
LIN {X 0,Y 435.462,Z 543.724,A -85,B 0,C 180,E1 -9286.888,E2 -9286.888} C_VEL
LIN {X 0,Y 436.539,Z 532.371,A -85,B 0,C 180,E1 -9288.22,E2 -9288.22} C_VEL
LIN {X 0,Y 437.525,Z 520.926,A -85,B 0,C 180,E1 -9289.347,E2 -9289.347} C_VEL
LIN {X 0,Y 438.697,Z 508.103,A -85,B 0,C 180,E1 -9290.391,E2 -9290.391} C_VEL
LIN {X 0,Y 439.536,Z 496.019,A -85,B 0,C 180,E1 -9291.208,E2 -9291.208} C_VEL
LIN {X 0,Y 440.407,Z 482.376,A -85,B 0,C 180,E1 -9291.945,E2 -9291.945} C_VEL
LIN {X 0,Y 441.117,Z 466.961,A -85,B 0,C 180,E1 -9292.573,E2 -9292.573} C_VEL
LIN {X 0,Y 441.557,Z 452.61,A -85,B 0,C 180,E1 -9292.982,E2 -9292.982} C_VEL
LIN {X 0,Y 443.387,Z 341.889,A -85,B 0,C 180,E1 -9294.831,E2 -9294.831} C_VEL
LIN {X 0,Y 443.692,Z 311.627,A -85,B 0,C 180,E1 -9295.343,E2 -9295.343} C_VEL
LIN {X 0,Y 442.183,Z 306.184,A -85,B 0,C 180,E1 -9295.533,E2 -9295.533} C_VEL
LIN {X 0,Y 434.434,Z 287.927,A -85,B 0,C 180,E1 -9296.368,E2 -9296.368} C_VEL
LIN {X 0,Y 432.371,Z 279.255,A -85,B 0,C 180,E1 -9298.25,E2 -9298.25} C_VEL
LIN {X 0,Y 432.3,Z 279.265,A -85,B 0,C 180,E1 -9301.347,E2 -9301.347} C_VEL
LIN {X 0,Y 432.321,Z 279.265,A -85,B 0,C 180,E1 -9304.678,E2 -9304.678} C_VEL
LIN {X 0,Y 432.32,Z 279.259,A -85,B 0,C 180,E1 -9308.151,E2 -9308.151} C_VEL
LIN {X 0,Y 432.301,Z 279.258,A -85,B 0,C 180,E1 -9311.801,E2 -9311.801} C_VEL
LIN {X 0,Y 432.33,Z 279.252,A -85,B 0,C 180,E1 -9314.347,E2 -9314.347} C_VEL
LIN {X 0,Y 432.298,Z 279.25,A -85,B 0,C 180,E1 -9317.018,E2 -9317.018} C_VEL
LIN {X 0,Y 432.285,Z 279.259,A -85,B 0,C 180,E1 -9319.828,E2 -9319.828} C_VEL
LIN {X 0,Y 432.29,Z 279.245,A -85,B 0,C 180,E1 -9323.02,E2 -9323.02} C_VEL
LIN {X 0,Y 432.327,Z 279.253,A -85,B 0,C 180,E1 -9326.002,E2 -9326.002} C_VEL
LIN {X 0,Y 432.328,Z 279.253,A -85,B 0,C 180,E1 -9329.493,E2 -9329.493} C_VEL
LIN {X 0,Y 432.312,Z 279.256,A -85,B 0,C 180,E1 -9331.872,E2 -9331.872} C_VEL
LIN {X 0,Y 432.319,Z 279.257,A -85,B 0,C 180,E1 -9334.997,E2 -9334.997} C_VEL
LIN {X 0,Y 432.348,Z 279.251,A -85,B 0,C 180,E1 -9338.045,E2 -9338.045} C_VEL
LIN {X 0,Y 432.341,Z 279.248,A -85,B 0,C 180,E1 -9341.027,E2 -9341.027} C_VEL
LIN {X 0,Y 432.383,Z 279.25,A -85,B 0,C 180,E1 -9343.959,E2 -9343.959} C_VEL
LIN {X 0,Y 432.457,Z 279.238,A -85,B 0,C 180,E1 -9347.803,E2 -9347.803} C_VEL
LIN {X 0,Y 432.445,Z 279.234,A -85,B 0,C 180,E1 -9351.589,E2 -9351.589} C_VEL
LIN {X 0,Y 432.546,Z 279.229,A -85,B 0,C 180,E1 -9354.405,E2 -9354.405} C_VEL
LIN {X 0,Y 432.6,Z 279.225,A -85,B 0,C 180,E1 -9358.138,E2 -9358.138} C_VEL
LIN {X 0,Y 432.545,Z 279.22,A -85,B 0,C 180,E1 -9360.931,E2 -9360.931} C_VEL
LIN {X 0,Y 432.564,Z 279.226,A -85,B 0,C 180,E1 -9362.794,E2 -9362.794} C_VEL
LIN {X 0,Y 432.576,Z 279.221,A -85,B 0,C 180,E1 -9365.594,E2 -9365.594} C_VEL
LIN {X 0,Y 432.461,Z 279.241,A -85,B 0,C 180,E1 -9368.41,E2 -9368.41} C_VEL
LIN {X 0,Y 432.458,Z 279.243,A -85,B 0,C 180,E1 -9372.197,E2 -9372.197} C_VEL
LIN {X 0,Y 432.429,Z 279.243,A -85,B 0,C 180,E1 -9376.039,E2 -9376.039} C_VEL
LIN {X 0,Y 432.385,Z 279.247,A -85,B 0,C 180,E1 -9379.485,E2 -9379.485} C_VEL
LIN {X 0,Y 432.316,Z 279.254,A -85,B 0,C 180,E1 -9382.964,E2 -9382.964} C_VEL
LIN {X 0,Y 432.337,Z 279.236,A -85,B 0,C 180,E1 -9385.002,E2 -9385.002} C_VEL
LIN {X 0,Y 432.346,Z 279.257,A -85,B 0,C 180,E1 -9388.126,E2 -9388.126} C_VEL
LIN {X 0,Y 432.319,Z 279.247,A -85,B 0,C 180,E1 -9391.346,E2 -9391.346} C_VEL
LIN {X 0,Y 432.338,Z 279.253,A -85,B 0,C 180,E1 -9394.677,E2 -9394.677} C_VEL
LIN {X 0,Y 432.337,Z 279.248,A -85,B 0,C 180,E1 -9398.15,E2 -9398.15} C_VEL
LIN {X 0,Y 432.331,Z 279.258,A -85,B 0,C 180,E1 -9401.602,E2 -9401.602} C_VEL
LIN {X 0,Y 432.332,Z 279.254,A -85,B 0,C 180,E1 -9404.347,E2 -9404.347} C_VEL
LIN {X 0,Y 432.318,Z 279.256,A -85,B 0,C 180,E1 -9407.016,E2 -9407.016} C_VEL
LIN {X 0,Y 432.331,Z 279.253,A -85,B 0,C 180,E1 -9409.821,E2 -9409.821} C_VEL
LIN {X 0,Y 432.306,Z 279.26,A -85,B 0,C 180,E1 -9413.022,E2 -9413.022} C_VEL
LIN {X 0,Y 432.358,Z 279.251,A -85,B 0,C 180,E1 -9415.997,E2 -9415.997} C_VEL
LIN {X 0,Y 432.351,Z 279.407,A -85,B 0,C 180,E1 -9417.318,E2 -9417.318} C_VEL
LIN {X 0,Y 436.571,Z 295.792,A -85,B 0,C 180,E1 -9420.377,E2 -9420.377} C_VEL
LIN {X 0,Y 438.338,Z 304.177,A -85,B 0,C 180,E1 -9421.864,E2 -9421.864} C_VEL
LIN {X 0,Y 437.463,Z 317.217,A -85,B 0,C 180,E1 -9423.875,E2 -9423.875} C_VEL
LIN {X 0,Y 443.363,Z 348.196,A -85,B 0,C 180,E1 -9424.788,E2 -9424.788} C_VEL
LIN {X 0,Y 441.477,Z 473.475,A -85,B 0,C 180,E1 -9426.859,E2 -9426.859} C_VEL
LIN {X 0,Y 441.07,Z 489.946,A -85,B 0,C 180,E1 -9427.208,E2 -9427.208} C_VEL
LIN {X 0,Y 440.275,Z 505.392,A -85,B 0,C 180,E1 -9427.719,E2 -9427.719} C_VEL
LIN {X 0,Y 439.463,Z 518.52,A -85,B 0,C 180,E1 -9428.319,E2 -9428.319} C_VEL
LIN {X 0,Y 438.476,Z 532.066,A -85,B 0,C 180,E1 -9429.107,E2 -9429.107} C_VEL
LIN {X 0,Y 437.27,Z 546.379,A -85,B 0,C 180,E1 -9430.152,E2 -9430.152} C_VEL
LIN {X 0,Y 436.112,Z 559.346,A -85,B 0,C 180,E1 -9431.32,E2 -9431.32} C_VEL
LIN {X 0,Y 434.95,Z 570.769,A -85,B 0,C 180,E1 -9432.551,E2 -9432.551} C_VEL
LIN {X 0,Y 434.173,Z 580.474,A -85,B 0,C 180,E1 -9433.786,E2 -9433.786} C_VEL
LIN {X 0,Y 433.225,Z 591.362,A -85,B 0,C 180,E1 -9435.437,E2 -9435.437} C_VEL
LIN {X 0,Y 432.388,Z 601.076,A -85,B 0,C 180,E1 -9437.222,E2 -9437.222} C_VEL
LIN {X 0,Y 432.059,Z 607.971,A -85,B 0,C 180,E1 -9438.744,E2 -9438.744} C_VEL
LIN {X 0,Y 431.564,Z 614.998,A -85,B 0,C 180,E1 -9440.628,E2 -9440.628} C_VEL
LIN {X 0,Y 431.341,Z 620.53,A -85,B 0,C 180,E1 -9442.511,E2 -9442.511} C_VEL
LIN {X 0,Y 431.222,Z 624.714,A -85,B 0,C 180,E1 -9444.389,E2 -9444.389} C_VEL
LIN {X 0,Y 431.169,Z 627.648,A -85,B 0,C 180,E1 -9446.262,E2 -9446.262} C_VEL
LIN {X 0,Y 431.215,Z 629.401,A -85,B 0,C 180,E1 -9448.132,E2 -9448.132} C_VEL
LIN {X 0,Y 431.19,Z 630,A -85,B 0,C 180,E1 -9450,E2 -9450} C_VEL
LIN {X 0,Y 431.215,Z 629.397,A -85,B 0,C 180,E1 -9451.868,E2 -9451.868} C_VEL
LIN {X 0,Y 431.169,Z 627.639,A -85,B 0,C 180,E1 -9453.739,E2 -9453.739} C_VEL
LIN {X 0,Y 431.212,Z 624.705,A -85,B 0,C 180,E1 -9455.612,E2 -9455.612} C_VEL
LIN {X 0,Y 431.328,Z 620.524,A -85,B 0,C 180,E1 -9457.49,E2 -9457.49} C_VEL
LIN {X 0,Y 431.556,Z 614.986,A -85,B 0,C 180,E1 -9459.373,E2 -9459.373} C_VEL
LIN {X 0,Y 432.05,Z 607.947,A -85,B 0,C 180,E1 -9461.257,E2 -9461.257} C_VEL
LIN {X 0,Y 432.577,Z 599.186,A -85,B 0,C 180,E1 -9463.148,E2 -9463.148} C_VEL
LIN {X 0,Y 433.345,Z 589.889,A -85,B 0,C 180,E1 -9464.8,E2 -9464.8} C_VEL
LIN {X 0,Y 434.165,Z 580.441,A -85,B 0,C 180,E1 -9466.215,E2 -9466.215} C_VEL
LIN {X 0,Y 435.238,Z 568.659,A -85,B 0,C 180,E1 -9467.693,E2 -9467.693} C_VEL
LIN {X 0,Y 436.404,Z 555.721,A -85,B 0,C 180,E1 -9469.034,E2 -9469.034} C_VEL
LIN {X 0,Y 437.656,Z 541.926,A -85,B 0,C 180,E1 -9470.198,E2 -9470.198} C_VEL
LIN {X 0,Y 438.756,Z 528.383,A -85,B 0,C 180,E1 -9471.126,E2 -9471.126} C_VEL
LIN {X 0,Y 439.72,Z 514.288,A -85,B 0,C 180,E1 -9471.893,E2 -9471.893} C_VEL
LIN {X 0,Y 440.615,Z 498.328,A -85,B 0,C 180,E1 -9472.539,E2 -9472.539} C_VEL
LIN {X 0,Y 441.28,Z 482.648,A -85,B 0,C 180,E1 -9472.967,E2 -9472.967} C_VEL
LIN {X 0,Y 443.365,Z 348.178,A -85,B 0,C 180,E1 -9475.207,E2 -9475.207} C_VEL
LIN {X 0,Y 437.436,Z 316.768,A -85,B 0,C 180,E1 -9476.153,E2 -9476.153} C_VEL
LIN {X 0,Y 438.337,Z 304.136,A -85,B 0,C 180,E1 -9478.136,E2 -9478.136} C_VEL
LIN {X 0,Y 435.75,Z 292.316,A -85,B 0,C 180,E1 -9480.246,E2 -9480.246} C_VEL
LIN {X 0,Y 432.352,Z 279.257,A -85,B 0,C 180,E1 -9482.718,E2 -9482.718} C_VEL
LIN {X 0,Y 432.34,Z 279.256,A -85,B 0,C 180,E1 -9485.818,E2 -9485.818} C_VEL
LIN {X 0,Y 432.324,Z 279.249,A -85,B 0,C 180,E1 -9489.346,E2 -9489.346} C_VEL
LIN {X 0,Y 432.326,Z 279.256,A -85,B 0,C 180,E1 -9491.799,E2 -9491.799} C_VEL
LIN {X 0,Y 432.336,Z 279.258,A -85,B 0,C 180,E1 -9494.348,E2 -9494.348} C_VEL
LIN {X 0,Y 432.323,Z 279.252,A -85,B 0,C 180,E1 -9497.016,E2 -9497.016} C_VEL
LIN {X 0,Y 432.336,Z 279.255,A -85,B 0,C 180,E1 -9499.821,E2 -9499.821} C_VEL
LIN {X 0,Y 432.308,Z 279.257,A -85,B 0,C 180,E1 -9503.022,E2 -9503.022} C_VEL
LIN {X 0,Y 432.363,Z 279.251,A -85,B 0,C 180,E1 -9505.997,E2 -9505.997} C_VEL
LIN {X 0,Y 432.35,Z 279.25,A -85,B 0,C 180,E1 -9509.49,E2 -9509.49} C_VEL
LIN {X 0,Y 432.351,Z 279.251,A -85,B 0,C 180,E1 -9511.875,E2 -9511.875} C_VEL
LIN {X 0,Y 432.382,Z 279.247,A -85,B 0,C 180,E1 -9515.539,E2 -9515.539} C_VEL
LIN {X 0,Y 432.355,Z 279.251,A -85,B 0,C 180,E1 -9519.046,E2 -9519.046} C_VEL
LIN {X 0,Y 432.377,Z 279.251,A -85,B 0,C 180,E1 -9522.011,E2 -9522.011} C_VEL
LIN {X 0,Y 432.399,Z 279.241,A -85,B 0,C 180,E1 -9524.927,E2 -9524.927} C_VEL
LIN {X 0,Y 432.464,Z 279.242,A -85,B 0,C 180,E1 -9527.804,E2 -9527.804} C_VEL
LIN {X 0,Y 432.467,Z 279.24,A -85,B 0,C 180,E1 -9531.59,E2 -9531.59} C_VEL
LIN {X 0,Y 432.577,Z 279.225,A -85,B 0,C 180,E1 -9534.406,E2 -9534.406} C_VEL
LIN {X 0,Y 432.6,Z 279.224,A -85,B 0,C 180,E1 -9538.138,E2 -9538.138} C_VEL
LIN {X 0,Y 432.625,Z 279.221,A -85,B 0,C 180,E1 -9540,E2 -9540} C_VEL
LIN {X 0,Y 432.574,Z 279.222,A -85,B 0,C 180,E1 -9542.794,E2 -9542.794} C_VEL
LIN {X 0,Y 432.515,Z 279.228,A -85,B 0,C 180,E1 -9546.531,E2 -9546.531} C_VEL
LIN {X 0,Y 432.429,Z 279.245,A -85,B 0,C 180,E1 -9549.354,E2 -9549.354} C_VEL
LIN {X 0,Y 432.436,Z 279.241,A -85,B 0,C 180,E1 -9552.803,E2 -9552.803} C_VEL
LIN {X 0,Y 432.361,Z 279.25,A -85,B 0,C 180,E1 -9556.453,E2 -9556.453} C_VEL
LIN {X 0,Y 432.318,Z 279.259,A -85,B 0,C 180,E1 -9559.962,E2 -9559.962} C_VEL
LIN {X 0,Y 432.306,Z 279.254,A -85,B 0,C 180,E1 -9562.965,E2 -9562.965} C_VEL
LIN {X 0,Y 432.309,Z 279.253,A -85,B 0,C 180,E1 -9566.036,E2 -9566.036} C_VEL
LIN {X 0,Y 432.318,Z 279.245,A -85,B 0,C 180,E1 -9569.189,E2 -9569.189} C_VEL
LIN {X 0,Y 432.308,Z 279.255,A -85,B 0,C 180,E1 -9572.444,E2 -9572.444} C_VEL
LIN {X 0,Y 432.333,Z 279.253,A -85,B 0,C 180,E1 -9575.818,E2 -9575.818} C_VEL
LIN {X 0,Y 432.314,Z 279.255,A -85,B 0,C 180,E1 -9578.709,E2 -9578.709} C_VEL
LIN {X 0,Y 432.303,Z 279.259,A -85,B 0,C 180,E1 -9581.801,E2 -9581.801} C_VEL
LIN {X 0,Y 432.312,Z 279.255,A -85,B 0,C 180,E1 -9584.35,E2 -9584.35} C_VEL
LIN {X 0,Y 432.259,Z 279.266,A -85,B 0,C 180,E1 -9587.025,E2 -9587.025} C_VEL
LIN {X 0,Y 432.289,Z 279.259,A -85,B 0,C 180,E1 -9589.828,E2 -9589.828} C_VEL
LIN {X 0,Y 432.295,Z 279.256,A -85,B 0,C 180,E1 -9593.02,E2 -9593.02} C_VEL
LIN {X 0,Y 432.332,Z 279.251,A -85,B 0,C 180,E1 -9596.002,E2 -9596.002} C_VEL
LIN {X 0,Y 432.333,Z 279.26,A -85,B 0,C 180,E1 -9599.493,E2 -9599.493} C_VEL
LIN {X 0,Y 432.378,Z 279.385,A -85,B 0,C 180,E1 -9601.909,E2 -9601.909} C_VEL
LIN {X 0,Y 434.41,Z 288.039,A -85,B 0,C 180,E1 -9603.74,E2 -9603.74} C_VEL
LIN {X 0,Y 442.665,Z 307.494,A -85,B 0,C 180,E1 -9604.616,E2 -9604.616} C_VEL
LIN {X 0,Y 443.802,Z 312.609,A -85,B 0,C 180,E1 -9604.777,E2 -9604.777} C_VEL
LIN {X 0,Y 442.193,Z 416.372,A -85,B 0,C 180,E1 -9606.495,E2 -9606.495} C_VEL
LIN {X 0,Y 441.546,Z 453.67,A -85,B 0,C 180,E1 -9607.14,E2 -9607.14} C_VEL
LIN {X 0,Y 441.005,Z 468.728,A -85,B 0,C 180,E1 -9607.58,E2 -9607.58} C_VEL
LIN {X 0,Y 440.597,Z 478.429,A -85,B 0,C 180,E1 -9607.971,E2 -9607.971} C_VEL
LIN {X 0,Y 439.716,Z 484.072,A -85,B 0,C 180,E1 -9608.199,E2 -9608.199} C_VEL
LIN {X 0,Y 436.463,Z 493.039,A -85,B 0,C 180,E1 -9608.533,E2 -9608.533} C_VEL
LIN {X 0,Y 433.138,Z 501.842,A -85,B 0,C 180,E1 -9608.937,E2 -9608.937} C_VEL
LIN {X 0,Y 432.138,Z 507.049,A -85,B 0,C 180,E1 -9609.277,E2 -9609.277} C_VEL
LIN {X 0,Y 430.93,Z 520.201,A -85,B 0,C 180,E1 -9610.344,E2 -9610.344} C_VEL
LIN {X 0,Y 429.832,Z 531.968,A -85,B 0,C 180,E1 -9611.502,E2 -9611.502} C_VEL
LIN {X 0,Y 428.697,Z 543.299,A -85,B 0,C 180,E1 -9612.837,E2 -9612.837} C_VEL
LIN {X 0,Y 427.688,Z 553.462,A -85,B 0,C 180,E1 -9614.268,E2 -9614.268} C_VEL
LIN {X 0,Y 426.674,Z 563.54,A -85,B 0,C 180,E1 -9615.963,E2 -9615.963} C_VEL
LIN {X 0,Y 425.951,Z 571.646,A -85,B 0,C 180,E1 -9617.614,E2 -9617.614} C_VEL
LIN {X 0,Y 425.238,Z 579.385,A -85,B 0,C 180,E1 -9619.525,E2 -9619.525} C_VEL
LIN {X 0,Y 424.76,Z 585.542,A -85,B 0,C 180,E1 -9621.436,E2 -9621.436} C_VEL
LIN {X 0,Y 424.454,Z 590.52,A -85,B 0,C 180,E1 -9623.446,E2 -9623.446} C_VEL
LIN {X 0,Y 424.25,Z 593.777,A -85,B 0,C 180,E1 -9625.248,E2 -9625.248} C_VEL
LIN {X 0,Y 424.26,Z 596.076,A -85,B 0,C 180,E1 -9627.151,E2 -9627.151} C_VEL
LIN {X 0,Y 424.112,Z 597.258,A -85,B 0,C 180,E1 -9629.05,E2 -9629.05} C_VEL
LIN {X 0,Y 424.113,Z 597.274,A -85,B 0,C 180,E1 -9630.949,E2 -9630.949} C_VEL
LIN {X 0,Y 424.261,Z 596.159,A -85,B 0,C 180,E1 -9632.848,E2 -9632.848} C_VEL
LIN {X 0,Y 424.247,Z 593.924,A -85,B 0,C 180,E1 -9634.751,E2 -9634.751} C_VEL
LIN {X 0,Y 424.456,Z 590.502,A -85,B 0,C 180,E1 -9636.655,E2 -9636.655} C_VEL
LIN {X 0,Y 424.751,Z 585.816,A -85,B 0,C 180,E1 -9638.564,E2 -9638.564} C_VEL
LIN {X 0,Y 425.21,Z 579.742,A -85,B 0,C 180,E1 -9640.475,E2 -9640.475} C_VEL
LIN {X 0,Y 425.909,Z 572.088,A -85,B 0,C 180,E1 -9642.387,E2 -9642.387} C_VEL
LIN {X 0,Y 426.606,Z 564.053,A -85,B 0,C 180,E1 -9644.039,E2 -9644.039} C_VEL
LIN {X 0,Y 427.644,Z 554.086,A -85,B 0,C 180,E1 -9645.733,E2 -9645.733} C_VEL
LIN {X 0,Y 428.644,Z 543.992,A -85,B 0,C 180,E1 -9647.165,E2 -9647.165} C_VEL
LIN {X 0,Y 429.883,Z 531.839,A -85,B 0,C 180,E1 -9648.605,E2 -9648.605} C_VEL
LIN {X 0,Y 430.988,Z 519.907,A -85,B 0,C 180,E1 -9649.777,E2 -9649.777} C_VEL
LIN {X 0,Y 432.17,Z 506.794,A -85,B 0,C 180,E1 -9650.838,E2 -9650.838} C_VEL
LIN {X 0,Y 433.079,Z 494.301,A -85,B 0,C 180,E1 -9651.665,E2 -9651.665} C_VEL
LIN {X 0,Y 433.986,Z 479.753,A -85,B 0,C 180,E1 -9652.427,E2 -9652.427} C_VEL
LIN {X 0,Y 434.691,Z 464.479,A -85,B 0,C 180,E1 -9653.02,E2 -9653.02} C_VEL
LIN {X 0,Y 435.156,Z 449.888,A -85,B 0,C 180,E1 -9653.403,E2 -9653.403} C_VEL
LIN {X 0,Y 436.71,Z 357.143,A -85,B 0,C 180,E1 -9654.969,E2 -9654.969} C_VEL
LIN {X 0,Y 437.263,Z 312.834,A -85,B 0,C 180,E1 -9655.725,E2 -9655.725} C_VEL
LIN {X 0,Y 435.974,Z 308.487,A -85,B 0,C 180,E1 -9655.886,E2 -9655.886} C_VEL
LIN {X 0,Y 427.243,Z 288.221,A -85,B 0,C 180,E1 -9656.846,E2 -9656.846} C_VEL
LIN {X 0,Y 425.29,Z 280.137,A -85,B 0,C 180,E1 -9658.635,E2 -9658.635} C_VEL
LIN {X 0,Y 425.245,Z 280.145,A -85,B 0,C 180,E1 -9661.928,E2 -9661.928} C_VEL
LIN {X 0,Y 425.289,Z 280.133,A -85,B 0,C 180,E1 -9665.336,E2 -9665.336} C_VEL
LIN {X 0,Y 425.274,Z 280.139,A -85,B 0,C 180,E1 -9668.901,E2 -9668.901} C_VEL
LIN {X 0,Y 425.253,Z 280.132,A -85,B 0,C 180,E1 -9672.655,E2 -9672.655} C_VEL
LIN {X 0,Y 425.281,Z 280.135,A -85,B 0,C 180,E1 -9675.283,E2 -9675.283} C_VEL
LIN {X 0,Y 425.242,Z 280.128,A -85,B 0,C 180,E1 -9678.617,E2 -9678.617} C_VEL
LIN {X 0,Y 425.265,Z 280.131,A -85,B 0,C 180,E1 -9682.304,E2 -9682.304} C_VEL
LIN {X 0,Y 425.28,Z 280.13,A -85,B 0,C 180,E1 -9685.815,E2 -9685.815} C_VEL
LIN {X 0,Y 425.282,Z 280.132,A -85,B 0,C 180,E1 -9689.24,E2 -9689.24} C_VEL
LIN {X 0,Y 425.239,Z 280.138,A -85,B 0,C 180,E1 -9692.434,E2 -9692.434} C_VEL
LIN {X 0,Y 425.315,Z 280.127,A -85,B 0,C 180,E1 -9695.6,E2 -9695.6} C_VEL
LIN {X 0,Y 425.279,Z 280.137,A -85,B 0,C 180,E1 -9698.681,E2 -9698.681} C_VEL
LIN {X 0,Y 425.282,Z 280.126,A -85,B 0,C 180,E1 -9701.7,E2 -9701.7} C_VEL
LIN {X 0,Y 425.298,Z 280.129,A -85,B 0,C 180,E1 -9704.669,E2 -9704.669} C_VEL
LIN {X 0,Y 425.41,Z 280.115,A -85,B 0,C 180,E1 -9707.598,E2 -9707.598} C_VEL
LIN {X 0,Y 425.394,Z 280.112,A -85,B 0,C 180,E1 -9711.449,E2 -9711.449} C_VEL
LIN {X 0,Y 425.504,Z 280.107,A -85,B 0,C 180,E1 -9714.312,E2 -9714.312} C_VEL
LIN {X 0,Y 425.569,Z 280.1,A -85,B 0,C 180,E1 -9718.107,E2 -9718.107} C_VEL
LIN {X 0,Y 425.507,Z 280.096,A -85,B 0,C 180,E1 -9720.946,E2 -9720.946} C_VEL
LIN {X 0,Y 425.519,Z 280.103,A -85,B 0,C 180,E1 -9722.84,E2 -9722.84} C_VEL
LIN {X 0,Y 425.53,Z 280.1,A -85,B 0,C 180,E1 -9725.687,E2 -9725.687} C_VEL
LIN {X 0,Y 425.406,Z 280.118,A -85,B 0,C 180,E1 -9728.551,E2 -9728.551} C_VEL
LIN {X 0,Y 425.411,Z 280.12,A -85,B 0,C 180,E1 -9732.402,E2 -9732.402} C_VEL
LIN {X 0,Y 425.386,Z 280.123,A -85,B 0,C 180,E1 -9736.312,E2 -9736.312} C_VEL
LIN {X 0,Y 425.327,Z 280.126,A -85,B 0,C 180,E1 -9739.635,E2 -9739.635} C_VEL
LIN {X 0,Y 425.303,Z 280.129,A -85,B 0,C 180,E1 -9743.365,E2 -9743.365} C_VEL
LIN {X 0,Y 425.3,Z 280.124,A -85,B 0,C 180,E1 -9746.498,E2 -9746.498} C_VEL
LIN {X 0,Y 425.284,Z 280.134,A -85,B 0,C 180,E1 -9749.72,E2 -9749.72} C_VEL
LIN {X 0,Y 425.28,Z 280.124,A -85,B 0,C 180,E1 -9753.048,E2 -9753.048} C_VEL
LIN {X 0,Y 425.281,Z 280.131,A -85,B 0,C 180,E1 -9755.929,E2 -9755.929} C_VEL
LIN {X 0,Y 425.299,Z 280.128,A -85,B 0,C 180,E1 -9759.044,E2 -9759.044} C_VEL
LIN {X 0,Y 425.273,Z 280.134,A -85,B 0,C 180,E1 -9762.653,E2 -9762.653} C_VEL
LIN {X 0,Y 425.259,Z 280.136,A -85,B 0,C 180,E1 -9766.044,E2 -9766.044} C_VEL
LIN {X 0,Y 425.272,Z 280.131,A -85,B 0,C 180,E1 -9768.622,E2 -9768.622} C_VEL
LIN {X 0,Y 425.304,Z 280.132,A -85,B 0,C 180,E1 -9771.102,E2 -9771.102} C_VEL
LIN {X 0,Y 425.299,Z 280.134,A -85,B 0,C 180,E1 -9774.664,E2 -9774.664} C_VEL
LIN {X 0,Y 425.309,Z 280.143,A -85,B 0,C 180,E1 -9776.884,E2 -9776.884} C_VEL
LIN {X 0,Y 429.648,Z 297.035,A -85,B 0,C 180,E1 -9780.106,E2 -9780.106} C_VEL
LIN {X 0,Y 431.555,Z 306.553,A -85,B 0,C 180,E1 -9781.818,E2 -9781.818} C_VEL
LIN {X 0,Y 430.759,Z 316.891,A -85,B 0,C 180,E1 -9783.436,E2 -9783.436} C_VEL
LIN {X 0,Y 436.88,Z 348.92,A -85,B 0,C 180,E1 -9784.404,E2 -9784.404} C_VEL
LIN {X 0,Y 435.27,Z 455.314,A -85,B 0,C 180,E1 -9786.193,E2 -9786.193} C_VEL
LIN {X 0,Y 434.678,Z 485.121,A -85,B 0,C 180,E1 -9786.727,E2 -9786.727} C_VEL
LIN {X 0,Y 433.943,Z 500.739,A -85,B 0,C 180,E1 -9787.195,E2 -9787.195} C_VEL
LIN {X 0,Y 433.066,Z 515.057,A -85,B 0,C 180,E1 -9787.806,E2 -9787.806} C_VEL
LIN {X 0,Y 432.111,Z 528.212,A -85,B 0,C 180,E1 -9788.534,E2 -9788.534} C_VEL
LIN {X 0,Y 430.993,Z 541.73,A -85,B 0,C 180,E1 -9789.477,E2 -9789.477} C_VEL
LIN {X 0,Y 429.657,Z 555.496,A -85,B 0,C 180,E1 -9790.657,E2 -9790.657} C_VEL
LIN {X 0,Y 428.447,Z 568.171,A -85,B 0,C 180,E1 -9791.988,E2 -9791.988} C_VEL
LIN {X 0,Y 427.307,Z 580.204,A -85,B 0,C 180,E1 -9793.518,E2 -9793.518} C_VEL
LIN {X 0,Y 426.258,Z 591.09,A -85,B 0,C 180,E1 -9795.194,E2 -9795.194} C_VEL
LIN {X 0,Y 425.434,Z 600.191,A -85,B 0,C 180,E1 -9796.878,E2 -9796.878} C_VEL
LIN {X 0,Y 425.026,Z 607.699,A -85,B 0,C 180,E1 -9798.556,E2 -9798.556} C_VEL
LIN {X 0,Y 424.501,Z 614.727,A -85,B 0,C 180,E1 -9800.471,E2 -9800.471} C_VEL
LIN {X 0,Y 424.278,Z 620.26,A -85,B 0,C 180,E1 -9802.385,E2 -9802.385} C_VEL
LIN {X 0,Y 424.138,Z 624.444,A -85,B 0,C 180,E1 -9804.295,E2 -9804.295} C_VEL
LIN {X 0,Y 424.079,Z 627.378,A -85,B 0,C 180,E1 -9806.2,E2 -9806.2} C_VEL
LIN {X 0,Y 424.141,Z 629.132,A -85,B 0,C 180,E1 -9808.101,E2 -9808.101} C_VEL
LIN {X 0,Y 424.105,Z 629.73,A -85,B 0,C 180,E1 -9810,E2 -9810} C_VEL
LIN {X 0,Y 424.141,Z 629.127,A -85,B 0,C 180,E1 -9811.9,E2 -9811.9} C_VEL
LIN {X 0,Y 424.079,Z 627.368,A -85,B 0,C 180,E1 -9813.801,E2 -9813.801} C_VEL
LIN {X 0,Y 424.125,Z 624.433,A -85,B 0,C 180,E1 -9815.706,E2 -9815.706} C_VEL
LIN {X 0,Y 424.269,Z 620.252,A -85,B 0,C 180,E1 -9817.616,E2 -9817.616} C_VEL
LIN {X 0,Y 424.493,Z 614.712,A -85,B 0,C 180,E1 -9819.53,E2 -9819.53} C_VEL
LIN {X 0,Y 425.014,Z 607.673,A -85,B 0,C 180,E1 -9821.446,E2 -9821.446} C_VEL
LIN {X 0,Y 425.578,Z 598.91,A -85,B 0,C 180,E1 -9823.368,E2 -9823.368} C_VEL
LIN {X 0,Y 426.401,Z 589.613,A -85,B 0,C 180,E1 -9825.046,E2 -9825.046} C_VEL
LIN {X 0,Y 427.297,Z 580.166,A -85,B 0,C 180,E1 -9826.483,E2 -9826.483} C_VEL
LIN {X 0,Y 428.467,Z 568.068,A -85,B 0,C 180,E1 -9828.019,E2 -9828.019} C_VEL
LIN {X 0,Y 429.662,Z 555.446,A -85,B 0,C 180,E1 -9829.344,E2 -9829.344} C_VEL
LIN {X 0,Y 430.973,Z 541.65,A -85,B 0,C 180,E1 -9830.525,E2 -9830.525} C_VEL
LIN {X 0,Y 432.098,Z 528.106,A -85,B 0,C 180,E1 -9831.467,E2 -9831.467} C_VEL
LIN {X 0,Y 433.106,Z 513.974,A -85,B 0,C 180,E1 -9832.247,E2 -9832.247} C_VEL
LIN {X 0,Y 433.998,Z 498.925,A -85,B 0,C 180,E1 -9832.871,E2 -9832.871} C_VEL
LIN {X 0,Y 434.719,Z 483.742,A -85,B 0,C 180,E1 -9833.303,E2 -9833.303} C_VEL
LIN {X 0,Y 436.965,Z 349.755,A -85,B 0,C 180,E1 -9835.57,E2 -9835.57} C_VEL
LIN {X 0,Y 431.138,Z 318.831,A -85,B 0,C 180,E1 -9836.497,E2 -9836.497} C_VEL
LIN {X 0,Y 430.708,Z 316.403,A -85,B 0,C 180,E1 -9836.607,E2 -9836.607} C_VEL
LIN {X 0,Y 431.525,Z 306.497,A -85,B 0,C 180,E1 -9838.185,E2 -9838.185} C_VEL
LIN {X 0,Y 429.647,Z 296.986,A -85,B 0,C 180,E1 -9839.894,E2 -9839.894} C_VEL
LIN {X 0,Y 425.312,Z 280.132,A -85,B 0,C 180,E1 -9843.117,E2 -9843.117} C_VEL
LIN {X 0,Y 425.267,Z 280.138,A -85,B 0,C 180,E1 -9846.509,E2 -9846.509} C_VEL
LIN {X 0,Y 425.279,Z 280.128,A -85,B 0,C 180,E1 -9849.04,E2 -9849.04} C_VEL
LIN {X 0,Y 425.285,Z 280.134,A -85,B 0,C 180,E1 -9851.957,E2 -9851.957} C_VEL
LIN {X 0,Y 425.287,Z 280.131,A -85,B 0,C 180,E1 -9855.284,E2 -9855.284} C_VEL
LIN {X 0,Y 425.278,Z 280.136,A -85,B 0,C 180,E1 -9858.622,E2 -9858.622} C_VEL
LIN {X 0,Y 425.299,Z 280.13,A -85,B 0,C 180,E1 -9861.102,E2 -9861.102} C_VEL
LIN {X 0,Y 425.302,Z 280.129,A -85,B 0,C 180,E1 -9864.664,E2 -9864.664} C_VEL
LIN {X 0,Y 425.269,Z 280.133,A -85,B 0,C 180,E1 -9868.074,E2 -9868.074} C_VEL
LIN {X 0,Y 425.318,Z 280.124,A -85,B 0,C 180,E1 -9871.367,E2 -9871.367} C_VEL
LIN {X 0,Y 425.275,Z 280.134,A -85,B 0,C 180,E1 -9874.553,E2 -9874.553} C_VEL
LIN {X 0,Y 425.288,Z 280.128,A -85,B 0,C 180,E1 -9876.634,E2 -9876.634} C_VEL
LIN {X 0,Y 425.3,Z 280.132,A -85,B 0,C 180,E1 -9879.695,E2 -9879.695} C_VEL
LIN {X 0,Y 425.344,Z 280.125,A -85,B 0,C 180,E1 -9882.698,E2 -9882.698} C_VEL
LIN {X 0,Y 425.352,Z 280.122,A -85,B 0,C 180,E1 -9885.65,E2 -9885.65} C_VEL
LIN {X 0,Y 425.353,Z 280.119,A -85,B 0,C 180,E1 -9888.564,E2 -9888.564} C_VEL
LIN {X 0,Y 425.411,Z 280.118,A -85,B 0,C 180,E1 -9891.449,E2 -9891.449} C_VEL
LIN {X 0,Y 425.531,Z 280.104,A -85,B 0,C 180,E1 -9894.313,E2 -9894.313} C_VEL
LIN {X 0,Y 425.569,Z 280.099,A -85,B 0,C 180,E1 -9898.107,E2 -9898.107} C_VEL
LIN {X 0,Y 425.577,Z 280.098,A -85,B 0,C 180,E1 -9900,E2 -9900} C_VEL
LIN {X 0,Y 425.529,Z 280.1,A -85,B 0,C 180,E1 -9902.84,E2 -9902.84} C_VEL
LIN {X 0,Y 425.477,Z 280.104,A -85,B 0,C 180,E1 -9906.64,E2 -9906.64} C_VEL
LIN {X 0,Y 425.39,Z 280.122,A -85,B 0,C 180,E1 -9909.51,E2 -9909.51} C_VEL
LIN {X 0,Y 425.398,Z 280.118,A -85,B 0,C 180,E1 -9912.903,E2 -9912.903} C_VEL
LIN {X 0,Y 425.318,Z 280.128,A -85,B 0,C 180,E1 -9916.583,E2 -9916.583} C_VEL
LIN {X 0,Y 425.3,Z 280.131,A -85,B 0,C 180,E1 -9919.623,E2 -9919.623} C_VEL
LIN {X 0,Y 425.289,Z 280.127,A -85,B 0,C 180,E1 -9922.339,E2 -9922.339} C_VEL
LIN {X 0,Y 425.255,Z 280.139,A -85,B 0,C 180,E1 -9925.448,E2 -9925.448} C_VEL
LIN {X 0,Y 425.299,Z 280.116,A -85,B 0,C 180,E1 -9928.857,E2 -9928.857} C_VEL
LIN {X 0,Y 425.249,Z 280.137,A -85,B 0,C 180,E1 -9931.928,E2 -9931.928} C_VEL
LIN {X 0,Y 425.292,Z 280.134,A -85,B 0,C 180,E1 -9935.337,E2 -9935.337} C_VEL
LIN {X 0,Y 425.267,Z 280.134,A -85,B 0,C 180,E1 -9938.902,E2 -9938.902} C_VEL
LIN {X 0,Y 425.245,Z 280.137,A -85,B 0,C 180,E1 -9941.95,E2 -9941.95} C_VEL
LIN {X 0,Y 425.252,Z 280.14,A -85,B 0,C 180,E1 -9945.288,E2 -9945.288} C_VEL
LIN {X 0,Y 425.246,Z 280.136,A -85,B 0,C 180,E1 -9948.617,E2 -9948.617} C_VEL
LIN {X 0,Y 425.269,Z 280.133,A -85,B 0,C 180,E1 -9952.304,E2 -9952.304} C_VEL
LIN {X 0,Y 425.284,Z 280.129,A -85,B 0,C 180,E1 -9955.815,E2 -9955.815} C_VEL
LIN {X 0,Y 425.286,Z 280.136,A -85,B 0,C 180,E1 -9959.24,E2 -9959.24} C_VEL
LIN {X 0,Y 425.299,Z 280.162,A -85,B 0,C 180,E1 -9961.5,E2 -9961.5} C_VEL
LIN {X 0,Y 427.29,Z 288.445,A -85,B 0,C 180,E1 -9963.269,E2 -9963.269} C_VEL
LIN {X 0,Y 436.468,Z 309.702,A -85,B 0,C 180,E1 -9964.264,E2 -9964.264} C_VEL
LIN {X 0,Y 437.334,Z 313.438,A -85,B 0,C 180,E1 -9964.387,E2 -9964.387} C_VEL
LIN {X 0,Y 435.714,Z 416.668,A -85,B 0,C 180,E1 -9966.123,E2 -9966.123} C_VEL
LIN {X 0,Y 435.042,Z 453.957,A -85,B 0,C 180,E1 -9966.779,E2 -9966.779} C_VEL
LIN {X 0,Y 434.481,Z 468.963,A -85,B 0,C 180,E1 -9967.222,E2 -9967.222} C_VEL
LIN {X 0,Y 433.745,Z 483.845,A -85,B 0,C 180,E1 -9967.857,E2 -9967.857} C_VEL
LIN {X 0,Y 432.751,Z 498.611,A -85,B 0,C 180,E1 -9968.692,E2 -9968.692} C_VEL
LIN {X 0,Y 432.138,Z 507.049,A -85,B 0,C 180,E1 -9969.277,E2 -9969.277} C_VEL
LIN {X 0,Y 431.123,Z 512.237,A -85,B 0,C 180,E1 -9969.638,E2 -9969.638} C_VEL
LIN {X 0,Y 424.674,Z 526.909,A -85,B 0,C 180,E1 -9970.687,E2 -9970.687} C_VEL
LIN {X 0,Y 423.227,Z 531.613,A -85,B 0,C 180,E1 -9971.129,E2 -9971.129} C_VEL
LIN {X 0,Y 423.01,Z 533.114,A -85,B 0,C 180,E1 -9971.296,E2 -9971.296} C_VEL
LIN {X 0,Y 421.895,Z 543.573,A -85,B 0,C 180,E1 -9972.551,E2 -9972.551} C_VEL
LIN {X 0,Y 420.818,Z 553.738,A -85,B 0,C 180,E1 -9974.004,E2 -9974.004} C_VEL
LIN {X 0,Y 419.76,Z 563.814,A -85,B 0,C 180,E1 -9975.727,E2 -9975.727} C_VEL
LIN {X 0,Y 418.995,Z 571.919,A -85,B 0,C 180,E1 -9977.405,E2 -9977.405} C_VEL
LIN {X 0,Y 418.212,Z 579.659,A -85,B 0,C 180,E1 -9979.347,E2 -9979.347} C_VEL
LIN {X 0,Y 417.711,Z 585.815,A -85,B 0,C 180,E1 -9981.29,E2 -9981.29} C_VEL
LIN {X 0,Y 417.393,Z 590.999,A -85,B 0,C 180,E1 -9983.431,E2 -9983.431} C_VEL
LIN {X 0,Y 417.185,Z 594.048,A -85,B 0,C 180,E1 -9985.168,E2 -9985.168} C_VEL
LIN {X 0,Y 417.174,Z 596.347,A -85,B 0,C 180,E1 -9987.103,E2 -9987.103} C_VEL
LIN {X 0,Y 417.033,Z 597.528,A -85,B 0,C 180,E1 -9989.034,E2 -9989.034} C_VEL
LIN {X 0,Y 417.034,Z 597.544,A -85,B 0,C 180,E1 -9990.965,E2 -9990.965} C_VEL
LIN {X 0,Y 417.174,Z 596.429,A -85,B 0,C 180,E1 -9992.897,E2 -9992.897} C_VEL
LIN {X 0,Y 417.182,Z 594.194,A -85,B 0,C 180,E1 -9994.831,E2 -9994.831} C_VEL
LIN {X 0,Y 417.404,Z 590.771,A -85,B 0,C 180,E1 -9996.768,E2 -9996.768} C_VEL
LIN {X 0,Y 417.7,Z 586.087,A -85,B 0,C 180,E1 -9998.709,E2 -9998.709} C_VEL
LIN {X 0,Y 418.186,Z 580.013,A -85,B 0,C 180,E1 -10000.653,E2 -10000.653} C_VEL
LIN {X 0,Y 418.949,Z 572.358,A -85,B 0,C 180,E1 -10002.596,E2 -10002.596} C_VEL
LIN {X 0,Y 419.715,Z 564.195,A -85,B 0,C 180,E1 -10004.299,E2 -10004.299} C_VEL
LIN {X 0,Y 420.772,Z 554.355,A -85,B 0,C 180,E1 -10005.997,E2 -10005.997} C_VEL
LIN {X 0,Y 421.833,Z 544.261,A -85,B 0,C 180,E1 -10007.451,E2 -10007.451} C_VEL
LIN {X 0,Y 423.118,Z 532.398,A -85,B 0,C 180,E1 -10008.879,E2 -10008.879} C_VEL
LIN {X 0,Y 424.325,Z 520.172,A -85,B 0,C 180,E1 -10010.101,E2 -10010.101} C_VEL
LIN {X 0,Y 425.523,Z 507.06,A -85,B 0,C 180,E1 -10011.179,E2 -10011.179} C_VEL
LIN {X 0,Y 426.501,Z 494.563,A -85,B 0,C 180,E1 -10012.017,E2 -10012.017} C_VEL
LIN {X 0,Y 427.461,Z 479.712,A -85,B 0,C 180,E1 -10012.803,E2 -10012.803} C_VEL
LIN {X 0,Y 428.173,Z 464.735,A -85,B 0,C 180,E1 -10013.391,E2 -10013.391} C_VEL
LIN {X 0,Y 428.664,Z 450.136,A -85,B 0,C 180,E1 -10013.779,E2 -10013.779} C_VEL
LIN {X 0,Y 430.65,Z 336.736,A -85,B 0,C 180,E1 -10015.72,E2 -10015.72} C_VEL
LIN {X 0,Y 430.885,Z 314.135,A -85,B 0,C 180,E1 -10016.115,E2 -10016.115} C_VEL
LIN {X 0,Y 428.861,Z 308.666,A -85,B 0,C 180,E1 -10016.35,E2 -10016.35} C_VEL
LIN {X 0,Y 420.108,Z 288.54,A -85,B 0,C 180,E1 -10017.334,E2 -10017.334} C_VEL
LIN {X 0,Y 418.243,Z 281.016,A -85,B 0,C 180,E1 -10019.055,E2 -10019.055} C_VEL
LIN {X 0,Y 418.229,Z 281.018,A -85,B 0,C 180,E1 -10022.529,E2 -10022.529} C_VEL
LIN {X 0,Y 418.247,Z 281.017,A -85,B 0,C 180,E1 -10024.842,E2 -10024.842} C_VEL
LIN {X 0,Y 418.232,Z 281.015,A -85,B 0,C 180,E1 -10028.444,E2 -10028.444} C_VEL
LIN {X 0,Y 418.216,Z 281.013,A -85,B 0,C 180,E1 -10032.236,E2 -10032.236} C_VEL
LIN {X 0,Y 418.232,Z 281.015,A -85,B 0,C 180,E1 -10035.108,E2 -10035.108} C_VEL
LIN {X 0,Y 418.214,Z 280.999,A -85,B 0,C 180,E1 -10037.763,E2 -10037.763} C_VEL
LIN {X 0,Y 418.224,Z 281.01,A -85,B 0,C 180,E1 -10041.555,E2 -10041.555} C_VEL
LIN {X 0,Y 418.245,Z 281.006,A -85,B 0,C 180,E1 -10045.157,E2 -10045.157} C_VEL
LIN {X 0,Y 418.229,Z 281.011,A -85,B 0,C 180,E1 -10047.47,E2 -10047.47} C_VEL
LIN {X 0,Y 418.255,Z 281.01,A -85,B 0,C 180,E1 -10050.898,E2 -10050.898} C_VEL
LIN {X 0,Y 418.215,Z 281.013,A -85,B 0,C 180,E1 -10054.092,E2 -10054.092} C_VEL
LIN {X 0,Y 418.222,Z 281.009,A -85,B 0,C 180,E1 -10057.263,E2 -10057.263} C_VEL
LIN {X 0,Y 418.248,Z 281.009,A -85,B 0,C 180,E1 -10060.362,E2 -10060.362} C_VEL
LIN {X 0,Y 418.277,Z 281.005,A -85,B 0,C 180,E1 -10063.403,E2 -10063.403} C_VEL
LIN {X 0,Y 418.345,Z 280.996,A -85,B 0,C 180,E1 -10066.999,E2 -10066.999} C_VEL
LIN {X 0,Y 418.325,Z 280.996,A -85,B 0,C 180,E1 -10070.328,E2 -10070.328} C_VEL
LIN {X 0,Y 418.436,Z 280.985,A -85,B 0,C 180,E1 -10073.248,E2 -10073.248} C_VEL
LIN {X 0,Y 418.318,Z 280.995,A -85,B 0,C 180,E1 -10075.181,E2 -10075.181} C_VEL
LIN {X 0,Y 418.538,Z 280.975,A -85,B 0,C 180,E1 -10078.075,E2 -10078.075} C_VEL
LIN {X 0,Y 418.471,Z 280.973,A -85,B 0,C 180,E1 -10080.962,E2 -10080.962} C_VEL
LIN {X 0,Y 418.476,Z 280.98,A -85,B 0,C 180,E1 -10082.888,E2 -10082.888} C_VEL
LIN {X 0,Y 418.487,Z 280.976,A -85,B 0,C 180,E1 -10085.783,E2 -10085.783} C_VEL
LIN {X 0,Y 418.375,Z 280.993,A -85,B 0,C 180,E1 -10088.695,E2 -10088.695} C_VEL
LIN {X 0,Y 418.312,Z 280.997,A -85,B 0,C 180,E1 -10091.631,E2 -10091.631} C_VEL
LIN {X 0,Y 418.3,Z 280.998,A -85,B 0,C 180,E1 -10094.597,E2 -10094.597} C_VEL
LIN {X 0,Y 418.284,Z 281.008,A -85,B 0,C 180,E1 -10097.604,E2 -10097.604} C_VEL
LIN {X 0,Y 418.248,Z 281.009,A -85,B 0,C 180,E1 -10100.663,E2 -10100.663} C_VEL
LIN {X 0,Y 418.283,Z 280.995,A -85,B 0,C 180,E1 -10103.781,E2 -10103.781} C_VEL
LIN {X 0,Y 418.225,Z 281.005,A -85,B 0,C 180,E1 -10107.048,E2 -10107.048} C_VEL
LIN {X 0,Y 418.241,Z 281.004,A -85,B 0,C 180,E1 -10110.272,E2 -10110.272} C_VEL
LIN {X 0,Y 418.247,Z 281.005,A -85,B 0,C 180,E1 -10113.677,E2 -10113.677} C_VEL
LIN {X 0,Y 418.239,Z 281.001,A -85,B 0,C 180,E1 -10117.224,E2 -10117.224} C_VEL
LIN {X 0,Y 418.253,Z 281.012,A -85,B 0,C 180,E1 -10119.682,E2 -10119.682} C_VEL
LIN {X 0,Y 418.228,Z 281.012,A -85,B 0,C 180,E1 -10122.321,E2 -10122.321} C_VEL
LIN {X 0,Y 418.234,Z 281.012,A -85,B 0,C 180,E1 -10125.109,E2 -10125.109} C_VEL
LIN {X 0,Y 418.238,Z 281.012,A -85,B 0,C 180,E1 -10127.767,E2 -10127.767} C_VEL
LIN {X 0,Y 418.251,Z 281.009,A -85,B 0,C 180,E1 -10130.62,E2 -10130.62} C_VEL
LIN {X 0,Y 418.243,Z 281.014,A -85,B 0,C 180,E1 -10133.976,E2 -10133.976} C_VEL
LIN {X 0,Y 418.293,Z 281.168,A -85,B 0,C 180,E1 -10136.488,E2 -10136.488} C_VEL
LIN {X 0,Y 422.724,Z 298.289,A -85,B 0,C 180,E1 -10139.828,E2 -10139.828} C_VEL
LIN {X 0,Y 424.727,Z 307.572,A -85,B 0,C 180,E1 -10141.542,E2 -10141.542} C_VEL
LIN {X 0,Y 424.052,Z 316.349,A -85,B 0,C 180,E1 -10142.972,E2 -10142.972} C_VEL
LIN {X 0,Y 430.41,Z 349.478,A -85,B 0,C 180,E1 -10144.005,E2 -10144.005} C_VEL
LIN {X 0,Y 429.17,Z 433.571,A -85,B 0,C 180,E1 -10145.447,E2 -10145.447} C_VEL
LIN {X 0,Y 428.23,Z 483.722,A -85,B 0,C 180,E1 -10146.324,E2 -10146.324} C_VEL
LIN {X 0,Y 427.462,Z 499.414,A -85,B 0,C 180,E1 -10146.785,E2 -10146.785} C_VEL
LIN {X 0,Y 426.471,Z 514.72,A -85,B 0,C 180,E1 -10147.44,E2 -10147.44} C_VEL
LIN {X 0,Y 425.478,Z 527.945,A -85,B 0,C 180,E1 -10148.183,E2 -10148.183} C_VEL
LIN {X 0,Y 424.291,Z 541.461,A -85,B 0,C 180,E1 -10149.138,E2 -10149.138} C_VEL
LIN {X 0,Y 422.898,Z 555.226,A -85,B 0,C 180,E1 -10150.335,E2 -10150.335} C_VEL
LIN {X 0,Y 421.606,Z 568.286,A -85,B 0,C 180,E1 -10151.732,E2 -10151.732} C_VEL
LIN {X 0,Y 420.45,Z 579.933,A -85,B 0,C 180,E1 -10153.242,E2 -10153.242} C_VEL
LIN {X 0,Y 419.33,Z 590.818,A -85,B 0,C 180,E1 -10154.943,E2 -10154.943} C_VEL
LIN {X 0,Y 418.474,Z 599.792,A -85,B 0,C 180,E1 -10156.628,E2 -10156.628} C_VEL
LIN {X 0,Y 417.954,Z 607.425,A -85,B 0,C 180,E1 -10158.359,E2 -10158.359} C_VEL
LIN {X 0,Y 417.423,Z 614.454,A -85,B 0,C 180,E1 -10160.308,E2 -10160.308} C_VEL
LIN {X 0,Y 417.185,Z 619.988,A -85,B 0,C 180,E1 -10162.255,E2 -10162.255} C_VEL
LIN {X 0,Y 417.057,Z 624.173,A -85,B 0,C 180,E1 -10164.197,E2 -10164.197} C_VEL
LIN {X 0,Y 416.993,Z 627.108,A -85,B 0,C 180,E1 -10166.135,E2 -10166.135} C_VEL
LIN {X 0,Y 417.067,Z 628.862,A -85,B 0,C 180,E1 -10168.069,E2 -10168.069} C_VEL
